LIN {X 0.123,Y -389.631,Z 435.593,A 0.000,B 0.000,C 90.000,E1 286.732} C_DIS
LIN {X -0.073,Y -402.281,Z 435.585,A 0.000,B 0.000,C 90.000,E1 285.371} C_DIS
LIN {X 0.165,Y -425.861,Z 435.572,A 0.000,B 0.000,C 90.000,E1 283.008} C_DIS
LIN {X -0.160,Y -433.525,Z 435.568,A 0.000,B 0.000,C 90.000,E1 282.299} C_DIS
LIN {X -0.184,Y -440.934,Z 435.564,A 0.000,B 0.000,C 90.000,E1 281.535} C_DIS
LIN {X 0.085,Y -448.117,Z 435.560,A 0.000,B 0.000,C 90.000,E1 280.715} C_DIS
LIN {X -0.168,Y -454.839,Z 435.555,A 0.000,B 0.000,C 90.000,E1 279.962} C_DIS
LIN {X 0.100,Y -461.020,Z 435.551,A 0.000,B 0.000,C 90.000,E1 279.151} C_DIS
LIN {X -0.034,Y -466.745,Z 435.547,A 0.000,B 0.000,C 90.000,E1 278.398} C_DIS
LIN {X 0.195,Y -473.496,Z 435.541,A 0.000,B 0.000,C 90.000,E1 277.352} C_DIS
LIN {X 0.113,Y -478.173,Z 435.537,A 0.000,B 0.000,C 90.000,E1 276.606} C_DIS
LIN {X 0.121,Y -482.372,Z 435.533,A 0.000,B 0.000,C 90.000,E1 275.853} C_DIS
LIN {X 0.118,Y -485.965,Z 435.528,A 0.000,B 0.000,C 90.000,E1 275.106} C_DIS
LIN {X 0.147,Y -488.810,Z 435.524,A 0.000,B 0.000,C 90.000,E1 274.359} C_DIS
LIN {X -0.139,Y -490.213,Z 435.522,A 0.000,B 0.000,C 90.000,E1 273.898} C_DIS
LIN {X 0.041,Y -491.202,Z 435.519,A 0.000,B 0.000,C 90.000,E1 273.383} C_DIS
LIN {X -0.232,Y -491.823,Z 435.516,A 0.000,B 0.000,C 90.000,E1 272.922} C_DIS
LIN {X -0.033,Y -492.111,Z 435.513,A 0.000,B 0.000,C 90.000,E1 272.407} C_DIS
LIN {X 0.172,Y -491.990,Z 435.511,A 0.000,B 0.000,C 90.000,E1 271.892} C_DIS
LIN {X -0.098,Y -491.492,Z 435.508,A 0.000,B 0.000,C 90.000,E1 271.432} C_DIS
LIN {X 0.107,Y -490.535,Z 435.505,A 0.000,B 0.000,C 90.000,E1 270.917} C_DIS
LIN {X -0.178,Y -489.067,Z 435.502,A 0.000,B 0.000,C 90.000,E1 270.458} C_DIS
LIN {X -0.128,Y -485.927,Z 435.498,A 0.000,B 0.000,C 90.000,E1 269.714} C_DIS
LIN {X 0.052,Y -483.029,Z 435.496,A 0.000,B 0.000,C 90.000,E1 269.198} C_DIS
LIN {X 0.210,Y -479.346,Z 435.493,A 0.000,B 0.000,C 90.000,E1 268.682} C_DIS
LIN {X -0.128,Y -474.646,Z 435.490,A 0.000,B 0.000,C 90.000,E1 268.224} C_DIS
LIN {X 0.188,Y -468.950,Z 435.487,A 0.000,B 0.000,C 90.000,E1 267.707} C_DIS
LIN {X -0.009,Y -462.615,Z 435.485,A 0.000,B 0.000,C 90.000,E1 267.306} C_DIS
LIN {X -0.137,Y -455.780,Z 435.483,A 0.000,B 0.000,C 90.000,E1 266.963} C_DIS
LIN {X -0.169,Y -448.676,Z 435.481,A 0.000,B 0.000,C 90.000,E1 266.674} C_DIS
LIN {X 0.179,Y -441.539,Z 435.480,A 0.000,B 0.000,C 90.000,E1 266.388} C_DIS
LIN {X -0.017,Y -433.742,Z 435.479,A 0.000,B 0.000,C 90.000,E1 266.216} C_DIS
LIN {X 0.183,Y -424.976,Z 435.478,A 0.000,B 0.000,C 90.000,E1 266.045} C_DIS
LIN {X -0.118,Y -414.468,Z 435.478,A 0.000,B 0.000,C 90.000,E1 265.988} C_DIS
LIN {X 0.107,Y -404.800,Z 435.477,A 0.000,B 0.000,C 90.000,E1 265.927} C_DIS
LIN {X 0.016,Y -180.918,Z 435.477,A 0.000,B 0.000,C 90.000,E1 265.927} C_DIS
LIN {X 0.049,Y -180.839,Z 435.472,A 0.000,B 0.000,C 90.000,E1 264.894} C_DIS
LIN {X -0.054,Y -178.880,Z 435.443,A 0.000,B 0.000,C 90.000,E1 259.690} C_DIS
LIN {X 0.022,Y -175.922,Z 435.414,A 0.000,B 0.000,C 90.000,E1 254.574} C_DIS
LIN {X -0.089,Y -174.621,Z 435.405,A 0.000,B 0.000,C 90.000,E1 252.906} C_DIS
LIN {X 0.004,Y -171.601,Z 435.381,A 0.000,B 0.000,C 90.000,E1 248.592} C_DIS
LIN {X -0.008,Y -167.824,Z 435.357,A 0.000,B 0.000,C 90.000,E1 244.280} C_DIS
LIN {X 0.010,Y -166.548,Z 435.347,A 0.000,B 0.000,C 90.000,E1 242.538} C_DIS
LIN {X -0.080,Y -162.545,Z 435.323,A 0.000,B 0.000,C 90.000,E1 238.201} C_DIS
LIN {X -0.019,Y -161.221,Z 435.313,A 0.000,B 0.000,C 90.000,E1 236.421} C_DIS
LIN {X 0.016,Y -157.229,Z 435.289,A 0.000,B 0.000,C 90.000,E1 231.984} C_DIS
LIN {X 0.039,Y -155.953,Z 435.279,A 0.000,B 0.000,C 90.000,E1 230.194} C_DIS
LIN {X -0.002,Y -152.206,Z 435.254,A 0.000,B 0.000,C 90.000,E1 225.729} C_DIS
LIN {X 0.018,Y -150.452,Z 435.239,A 0.000,B 0.000,C 90.000,E1 223.014} C_DIS
LIN {X 0.045,Y -147.177,Z 435.214,A 0.000,B 0.000,C 90.000,E1 218.463} C_DIS
LIN {X 0.012,Y -145.194,Z 435.193,A 0.000,B 0.000,C 90.000,E1 214.818} C_DIS
LIN {X 0.046,Y -142.335,Z 435.163,A 0.000,B 0.000,C 90.000,E1 209.283} C_DIS
LIN {X -0.025,Y -141.724,Z 435.153,A 0.000,B 0.000,C 90.000,E1 207.462} C_DIS
LIN {X -0.042,Y -139.478,Z 435.116,A 0.000,B 0.000,C 90.000,E1 200.972} C_DIS
LIN {X -0.054,Y -138.976,Z 435.101,A 0.000,B 0.000,C 90.000,E1 198.181} C_DIS
LIN {X 0.068,Y -138.332,Z 435.054,A 0.000,B 0.000,C 90.000,E1 189.726} C_DIS
LIN {X -0.068,Y -139.431,Z 435.007,A 0.000,B 0.000,C 90.000,E1 181.375} C_DIS
LIN {X 0.012,Y -140.958,Z 434.976,A 0.000,B 0.000,C 90.000,E1 175.755} C_DIS
LIN {X -0.038,Y -142.714,Z 434.956,A 0.000,B 0.000,C 90.000,E1 172.064} C_DIS
LIN {X 0.062,Y -145.091,Z 434.930,A 0.000,B 0.000,C 90.000,E1 167.409} C_DIS
LIN {X 0.057,Y -147.716,Z 434.910,A 0.000,B 0.000,C 90.000,E1 163.740} C_DIS
LIN {X -0.002,Y -150.372,Z 434.890,A 0.000,B 0.000,C 90.000,E1 160.115} C_DIS
LIN {X 0.016,Y -153.801,Z 434.869,A 0.000,B 0.000,C 90.000,E1 156.485} C_DIS
LIN {X 0.076,Y -157.213,Z 434.849,A 0.000,B 0.000,C 90.000,E1 152.871} C_DIS
LIN {X 0.017,Y -161.377,Z 434.830,A 0.000,B 0.000,C 90.000,E1 149.331} C_DIS
LIN {X 0.028,Y -165.580,Z 434.810,A 0.000,B 0.000,C 90.000,E1 145.801} C_DIS
LIN {X 0.015,Y -170.500,Z 434.791,A 0.000,B 0.000,C 90.000,E1 142.316} C_DIS
LIN {X 0.059,Y -175.380,Z 434.772,A 0.000,B 0.000,C 90.000,E1 138.852} C_DIS
LIN {X -0.079,Y -181.005,Z 434.753,A 0.000,B 0.000,C 90.000,E1 135.486} C_DIS
LIN {X 0.046,Y -186.434,Z 434.734,A 0.000,B 0.000,C 90.000,E1 132.081} C_DIS
LIN {X 0.115,Y -191.060,Z 434.720,A 0.000,B 0.000,C 90.000,E1 129.564} C_DIS
LIN {X 0.004,Y -195.867,Z 434.705,A 0.000,B 0.000,C 90.000,E1 126.824} C_DIS
LIN {X 0.135,Y -294.379,Z 434.705,A 0.000,B 0.000,C 90.000,E1 126.790} C_DIS
LIN {X -0.008,Y -296.001,Z 434.704,A 0.000,B 0.000,C 90.000,E1 126.790} C_DIS
LIN {X 0.056,Y -300.860,Z 434.703,A 0.000,B 0.000,C 90.000,E1 126.537} C_DIS
LIN {X 0.058,Y -303.494,Z 434.702,A 0.000,B 0.000,C 90.000,E1 126.297} C_DIS
LIN {X -0.117,Y -307.272,Z 434.699,A 0.000,B 0.000,C 90.000,E1 125.804} C_DIS
LIN {X 0.085,Y -308.927,Z 434.697,A 0.000,B 0.000,C 90.000,E1 125.438} C_DIS
LIN {X 0.109,Y -310.232,Z 434.695,A 0.000,B 0.000,C 90.000,E1 125.105} C_DIS
LIN {X -0.103,Y -322.084,Z 434.675,A 0.000,B 0.000,C 90.000,E1 121.592} C_DIS
LIN {X -0.105,Y -333.198,Z 434.660,A 0.000,B 0.000,C 90.000,E1 118.743} C_DIS
LIN {X 0.047,Y -345.725,Z 434.644,A 0.000,B 0.000,C 90.000,E1 115.924} C_DIS
LIN {X -0.096,Y -358.139,Z 434.631,A 0.000,B 0.000,C 90.000,E1 113.515} C_DIS
LIN {X 0.113,Y -371.851,Z 434.617,A 0.000,B 0.000,C 90.000,E1 111.099} C_DIS
LIN {X 0.056,Y -386.960,Z 434.604,A 0.000,B 0.000,C 90.000,E1 108.779} C_DIS
LIN {X 0.125,Y -403.577,Z 434.592,A 0.000,B 0.000,C 90.000,E1 106.496} C_DIS
LIN {X -0.010,Y -421.825,Z 434.579,A 0.000,B 0.000,C 90.000,E1 104.300} C_DIS
LIN {X -0.034,Y -441.588,Z 434.568,A 0.000,B 0.000,C 90.000,E1 102.175} C_DIS
LIN {X 0.112,Y -462.024,Z 434.557,A 0.000,B 0.000,C 90.000,E1 100.197} C_DIS
LIN {X -0.173,Y -485.514,Z 434.546,A 0.000,B 0.000,C 90.000,E1 98.219} C_DIS
LIN {X 0.009,Y -489.050,Z 434.543,A 0.000,B 0.000,C 90.000,E1 97.757} C_DIS
LIN {X -0.167,Y -490.369,Z 434.542,A 0.000,B 0.000,C 90.000,E1 97.530} C_DIS
LIN {X 0.207,Y -491.341,Z 434.540,A 0.000,B 0.000,C 90.000,E1 97.239} C_DIS
LIN {X -0.056,Y -492.420,Z 434.538,A 0.000,B 0.000,C 90.000,E1 96.777} C_DIS
LIN {X 0.177,Y -492.489,Z 434.535,A 0.000,B 0.000,C 90.000,E1 96.258} C_DIS
LIN {X -0.075,Y -491.558,Z 434.532,A 0.000,B 0.000,C 90.000,E1 95.796} C_DIS
LIN {X 0.161,Y -489.465,Z 434.529,A 0.000,B 0.000,C 90.000,E1 95.277} C_DIS
LIN {X 0.011,Y -487.840,Z 434.528,A 0.000,B 0.000,C 90.000,E1 95.049} C_DIS
LIN {X -0.226,Y -478.097,Z 434.521,A 0.000,B 0.000,C 90.000,E1 93.841} C_DIS
LIN {X 0.010,Y -456.548,Z 434.506,A 0.000,B 0.000,C 90.000,E1 91.031} C_DIS
LIN {X 0.172,Y -444.184,Z 434.496,A 0.000,B 0.000,C 90.000,E1 89.198} C_DIS
LIN {X -0.022,Y -429.185,Z 434.482,A 0.000,B 0.000,C 90.000,E1 86.846} C_DIS
LIN {X -0.046,Y -413.302,Z 434.467,A 0.000,B 0.000,C 90.000,E1 84.147} C_DIS
LIN {X -0.128,Y -400.978,Z 434.455,A 0.000,B 0.000,C 90.000,E1 81.951} C_DIS
LIN {X -0.101,Y -390.349,Z 434.444,A 0.000,B 0.000,C 90.000,E1 79.982} C_DIS
LIN {X 0.180,Y -381.300,Z 434.435,A 0.000,B 0.000,C 90.000,E1 78.229} C_DIS
LIN {X 0.081,Y -366.697,Z 434.419,A 0.000,B 0.000,C 90.000,E1 75.338} C_DIS
LIN {X 0.065,Y -350.448,Z 434.399,A 0.000,B 0.000,C 90.000,E1 71.764} C_DIS
LIN {X 0.015,Y -339.131,Z 434.384,A 0.000,B 0.000,C 90.000,E1 69.028} C_DIS
LIN {X 0.059,Y -329.454,Z 434.370,A 0.000,B 0.000,C 90.000,E1 66.538} C_DIS
LIN {X -0.056,Y -318.843,Z 434.354,A 0.000,B 0.000,C 90.000,E1 63.717} C_DIS
LIN {X 0.040,Y -309.658,Z 434.340,A 0.000,B 0.000,C 90.000,E1 61.129} C_DIS
LIN {X -0.012,Y -298.573,Z 434.321,A 0.000,B 0.000,C 90.000,E1 57.867} C_DIS
LIN {X 0.030,Y -288.435,Z 434.303,A 0.000,B 0.000,C 90.000,E1 54.529} C_DIS
LIN {X 0.017,Y -280.852,Z 434.288,A 0.000,B 0.000,C 90.000,E1 51.823} C_DIS
LIN {X 0.115,Y -275.170,Z 434.276,A 0.000,B 0.000,C 90.000,E1 49.747} C_DIS
LIN {X -0.105,Y -269.235,Z 434.265,A 0.000,B 0.000,C 90.000,E1 47.715} C_DIS
LIN {X 0.105,Y -263.070,Z 434.253,A 0.000,B 0.000,C 90.000,E1 45.567} C_DIS
LIN {X 0.012,Y -256.793,Z 434.241,A 0.000,B 0.000,C 90.000,E1 43.461} C_DIS
LIN {X 0.001,Y -250.333,Z 434.229,A 0.000,B 0.000,C 90.000,E1 41.310} C_DIS
LIN {X 0.045,Y -239.769,Z 434.209,A 0.000,B 0.000,C 90.000,E1 37.649} C_DIS
LIN {X -0.031,Y -231.877,Z 434.193,A 0.000,B 0.000,C 90.000,E1 34.692} C_DIS
LIN {X -0.045,Y -224.697,Z 434.176,A 0.000,B 0.000,C 90.000,E1 31.671} C_DIS
LIN {X -0.090,Y -218.311,Z 434.159,A 0.000,B 0.000,C 90.000,E1 28.615} C_DIS
LIN {X 0.069,Y -212.674,Z 434.142,A 0.000,B 0.000,C 90.000,E1 25.463} C_DIS
LIN {X 0.029,Y -206.563,Z 434.120,A 0.000,B 0.000,C 90.000,E1 21.535} C_DIS
LIN {X -0.102,Y -201.340,Z 434.098,A 0.000,B 0.000,C 90.000,E1 17.583} C_DIS
LIN {X -0.052,Y -197.150,Z 434.075,A 0.000,B 0.000,C 90.000,E1 13.536} C_DIS
LIN {X 0.032,Y -193.335,Z 434.048,A 0.000,B 0.000,C 90.000,E1 8.624} C_DIS
LIN {X -0.006,Y -190.457,Z 434.011,A 0.000,B 0.000,C 90.000,E1 2.064} C_DIS
LIN {X -0.008,Y -191.173,Z 433.961,A 0.000,B 0.000,C 90.000,E1 352.932} C_DIS
LIN {X 0.006,Y -194.242,Z 433.929,A 0.000,B 0.000,C 90.000,E1 347.173} C_DIS
LIN {X -0.103,Y -198.351,Z 433.902,A 0.000,B 0.000,C 90.000,E1 342.308} C_DIS
LIN {X 0.010,Y -202.852,Z 433.879,A 0.000,B 0.000,C 90.000,E1 338.230} C_DIS
LIN {X 0.006,Y -208.404,Z 433.857,A 0.000,B 0.000,C 90.000,E1 334.229} C_DIS
LIN {X 0.083,Y -214.790,Z 433.835,A 0.000,B 0.000,C 90.000,E1 330.255} C_DIS
LIN {X 0.018,Y -221.686,Z 433.813,A 0.000,B 0.000,C 90.000,E1 326.373} C_DIS
LIN {X -0.082,Y -229.246,Z 433.792,A 0.000,B 0.000,C 90.000,E1 322.557} C_DIS
LIN {X -0.060,Y -237.792,Z 433.771,A 0.000,B 0.000,C 90.000,E1 318.771} C_DIS
LIN {X 0.032,Y -246.477,Z 433.752,A 0.000,B 0.000,C 90.000,E1 315.405} C_DIS
LIN {X -0.148,Y -255.172,Z 433.736,A 0.000,B 0.000,C 90.000,E1 312.528} C_DIS
LIN {X -0.018,Y -266.116,Z 433.718,A 0.000,B 0.000,C 90.000,E1 309.277} C_DIS
LIN {X -0.072,Y -278.087,Z 433.701,A 0.000,B 0.000,C 90.000,E1 306.137} C_DIS
LIN {X 0.042,Y -289.473,Z 433.685,A 0.000,B 0.000,C 90.000,E1 303.372} C_DIS
LIN {X -0.084,Y -304.390,Z 433.667,A 0.000,B 0.000,C 90.000,E1 300.050} C_DIS
LIN {X -0.090,Y -320.673,Z 433.649,A 0.000,B 0.000,C 90.000,E1 296.796} C_DIS
LIN {X -0.121,Y -336.820,Z 433.633,A 0.000,B 0.000,C 90.000,E1 293.951} C_DIS
LIN {X 0.023,Y -353.039,Z 433.619,A 0.000,B 0.000,C 90.000,E1 291.461} C_DIS
LIN {X -0.137,Y -370.722,Z 433.606,A 0.000,B 0.000,C 90.000,E1 289.087} C_DIS
LIN {X 0.026,Y -389.759,Z 433.593,A 0.000,B 0.000,C 90.000,E1 286.732} C_DIS
LIN {X 0.144,Y -404.944,Z 433.584,A 0.000,B 0.000,C 90.000,E1 285.064} C_DIS
LIN {X 0.164,Y -425.900,Z 433.572,A 0.000,B 0.000,C 90.000,E1 283.008} C_DIS
LIN {X -0.156,Y -433.580,Z 433.568,A 0.000,B 0.000,C 90.000,E1 282.299} C_DIS
LIN {X 0.043,Y -443.390,Z 433.563,A 0.000,B 0.000,C 90.000,E1 281.243} C_DIS
LIN {X -0.227,Y -450.440,Z 433.558,A 0.000,B 0.000,C 90.000,E1 280.489} C_DIS
LIN {X 0.076,Y -456.998,Z 433.554,A 0.000,B 0.000,C 90.000,E1 279.670} C_DIS
LIN {X -0.096,Y -463.001,Z 433.549,A 0.000,B 0.000,C 90.000,E1 278.916} C_DIS
LIN {X -0.212,Y -468.492,Z 433.545,A 0.000,B 0.000,C 90.000,E1 278.163} C_DIS
LIN {X -0.028,Y -475.101,Z 433.540,A 0.000,B 0.000,C 90.000,E1 277.125} C_DIS
LIN {X -0.047,Y -479.630,Z 433.535,A 0.000,B 0.000,C 90.000,E1 276.372} C_DIS
LIN {X -0.075,Y -483.657,Z 433.531,A 0.000,B 0.000,C 90.000,E1 275.625} C_DIS
LIN {X -0.068,Y -487.018,Z 433.527,A 0.000,B 0.000,C 90.000,E1 274.878} C_DIS
LIN {X 0.131,Y -488.800,Z 433.524,A 0.000,B 0.000,C 90.000,E1 274.359} C_DIS
LIN {X -0.155,Y -490.188,Z 433.522,A 0.000,B 0.000,C 90.000,E1 273.898} C_DIS
LIN {X 0.026,Y -491.171,Z 433.519,A 0.000,B 0.000,C 90.000,E1 273.383} C_DIS
LIN {X 0.244,Y -491.813,Z 433.516,A 0.000,B 0.000,C 90.000,E1 272.865} C_DIS
LIN {X -0.049,Y -492.116,Z 433.513,A 0.000,B 0.000,C 90.000,E1 272.407} C_DIS
LIN {X 0.156,Y -492.028,Z 433.511,A 0.000,B 0.000,C 90.000,E1 271.892} C_DIS
LIN {X -0.114,Y -491.524,Z 433.508,A 0.000,B 0.000,C 90.000,E1 271.432} C_DIS
LIN {X 0.092,Y -490.557,Z 433.505,A 0.000,B 0.000,C 90.000,E1 270.917} C_DIS
LIN {X -0.194,Y -489.104,Z 433.502,A 0.000,B 0.000,C 90.000,E1 270.458} C_DIS
LIN {X 0.005,Y -487.130,Z 433.500,A 0.000,B 0.000,C 90.000,E1 269.943} C_DIS
LIN {X 0.194,Y -484.575,Z 433.497,A 0.000,B 0.000,C 90.000,E1 269.427} C_DIS
LIN {X -0.120,Y -481.344,Z 433.494,A 0.000,B 0.000,C 90.000,E1 268.969} C_DIS
LIN {X 0.031,Y -477.139,Z 433.491,A 0.000,B 0.000,C 90.000,E1 268.453} C_DIS
LIN {X -0.143,Y -474.692,Z 433.490,A 0.000,B 0.000,C 90.000,E1 268.224} C_DIS
LIN {X 0.172,Y -469.070,Z 433.487,A 0.000,B 0.000,C 90.000,E1 267.707} C_DIS
LIN {X 0.169,Y -465.857,Z 433.486,A 0.000,B 0.000,C 90.000,E1 267.478} C_DIS
LIN {X 0.214,Y -459.156,Z 433.484,A 0.000,B 0.000,C 90.000,E1 267.078} C_DIS
LIN {X -0.067,Y -452.119,Z 433.482,A 0.000,B 0.000,C 90.000,E1 266.788} C_DIS
LIN {X 0.105,Y -445.016,Z 433.481,A 0.000,B 0.000,C 90.000,E1 266.502} C_DIS
LIN {X 0.191,Y -437.456,Z 433.479,A 0.000,B 0.000,C 90.000,E1 266.274} C_DIS
LIN {X 0.206,Y -429.445,Z 433.478,A 0.000,B 0.000,C 90.000,E1 266.102} C_DIS
LIN {X 0.123,Y -418.947,Z 433.478,A 0.000,B 0.000,C 90.000,E1 265.988} C_DIS
LIN {X 0.134,Y -408.679,Z 433.477,A 0.000,B 0.000,C 90.000,E1 265.927} C_DIS
LIN {X 0.028,Y -180.917,Z 433.477,A 0.000,B 0.000,C 90.000,E1 265.927} C_DIS
LIN {X 0.059,Y -180.839,Z 433.472,A 0.000,B 0.000,C 90.000,E1 264.894} C_DIS
LIN {X -0.044,Y -178.881,Z 433.443,A 0.000,B 0.000,C 90.000,E1 259.690} C_DIS
LIN {X 0.033,Y -175.924,Z 433.414,A 0.000,B 0.000,C 90.000,E1 254.574} C_DIS
LIN {X -0.022,Y -175.361,Z 433.410,A 0.000,B 0.000,C 90.000,E1 253.740} C_DIS
LIN {X 0.037,Y -172.140,Z 433.386,A 0.000,B 0.000,C 90.000,E1 249.444} C_DIS
LIN {X 0.014,Y -171.604,Z 433.381,A 0.000,B 0.000,C 90.000,E1 248.592} C_DIS
LIN {X 0.002,Y -167.827,Z 433.357,A 0.000,B 0.000,C 90.000,E1 244.280} C_DIS
LIN {X 0.020,Y -166.552,Z 433.347,A 0.000,B 0.000,C 90.000,E1 242.538} C_DIS
LIN {X -0.070,Y -162.547,Z 433.323,A 0.000,B 0.000,C 90.000,E1 238.201} C_DIS
LIN {X -0.010,Y -161.225,Z 433.313,A 0.000,B 0.000,C 90.000,E1 236.421} C_DIS
LIN {X 0.025,Y -157.231,Z 433.289,A 0.000,B 0.000,C 90.000,E1 231.984} C_DIS
LIN {X 0.048,Y -155.955,Z 433.279,A 0.000,B 0.000,C 90.000,E1 230.194} C_DIS
LIN {X 0.007,Y -152.209,Z 433.254,A 0.000,B 0.000,C 90.000,E1 225.729} C_DIS
LIN {X 0.028,Y -150.454,Z 433.239,A 0.000,B 0.000,C 90.000,E1 223.014} C_DIS
LIN {X 0.054,Y -147.179,Z 433.214,A 0.000,B 0.000,C 90.000,E1 218.463} C_DIS
LIN {X 0.021,Y -145.197,Z 433.193,A 0.000,B 0.000,C 90.000,E1 214.818} C_DIS
LIN {X 0.056,Y -142.336,Z 433.163,A 0.000,B 0.000,C 90.000,E1 209.283} C_DIS
LIN {X -0.015,Y -141.724,Z 433.153,A 0.000,B 0.000,C 90.000,E1 207.462} C_DIS
LIN {X -0.033,Y -139.479,Z 433.116,A 0.000,B 0.000,C 90.000,E1 200.972} C_DIS
LIN {X -0.044,Y -138.977,Z 433.101,A 0.000,B 0.000,C 90.000,E1 198.181} C_DIS
LIN {X 0.077,Y -138.331,Z 433.054,A 0.000,B 0.000,C 90.000,E1 189.726} C_DIS
LIN {X -0.059,Y -139.431,Z 433.008,A 0.000,B 0.000,C 90.000,E1 181.375} C_DIS
LIN {X 0.020,Y -140.956,Z 432.976,A 0.000,B 0.000,C 90.000,E1 175.755} C_DIS
LIN {X -0.029,Y -142.713,Z 432.956,A 0.000,B 0.000,C 90.000,E1 172.064} C_DIS
LIN {X 0.070,Y -145.089,Z 432.930,A 0.000,B 0.000,C 90.000,E1 167.409} C_DIS
LIN {X 0.066,Y -147.713,Z 432.910,A 0.000,B 0.000,C 90.000,E1 163.740} C_DIS
LIN {X 0.008,Y -150.370,Z 432.890,A 0.000,B 0.000,C 90.000,E1 160.115} C_DIS
LIN {X 0.025,Y -153.797,Z 432.869,A 0.000,B 0.000,C 90.000,E1 156.485} C_DIS
LIN {X 0.086,Y -157.210,Z 432.849,A 0.000,B 0.000,C 90.000,E1 152.871} C_DIS
LIN {X 0.028,Y -161.373,Z 432.830,A 0.000,B 0.000,C 90.000,E1 149.331} C_DIS
LIN {X 0.039,Y -165.575,Z 432.810,A 0.000,B 0.000,C 90.000,E1 145.801} C_DIS
LIN {X 0.025,Y -170.495,Z 432.791,A 0.000,B 0.000,C 90.000,E1 142.316} C_DIS
LIN {X 0.070,Y -175.375,Z 432.772,A 0.000,B 0.000,C 90.000,E1 138.852} C_DIS
LIN {X -0.067,Y -180.999,Z 432.753,A 0.000,B 0.000,C 90.000,E1 135.486} C_DIS
LIN {X 0.057,Y -186.427,Z 432.734,A 0.000,B 0.000,C 90.000,E1 132.081} C_DIS
LIN {X 0.004,Y -191.054,Z 432.720,A 0.000,B 0.000,C 90.000,E1 129.600} C_DIS
LIN {X -0.067,Y -195.970,Z 432.704,A 0.000,B 0.000,C 90.000,E1 126.790} C_DIS
LIN {X -0.136,Y -294.358,Z 432.704,A 0.000,B 0.000,C 90.000,E1 126.790} C_DIS
LIN {X -0.078,Y -296.347,Z 432.704,A 0.000,B 0.000,C 90.000,E1 126.744} C_DIS
LIN {X 0.087,Y -300.646,Z 432.703,A 0.000,B 0.000,C 90.000,E1 126.503} C_DIS
LIN {X 0.076,Y -303.088,Z 432.702,A 0.000,B 0.000,C 90.000,E1 126.297} C_DIS
LIN {X 0.046,Y -306.923,Z 432.699,A 0.000,B 0.000,C 90.000,E1 125.804} C_DIS
LIN {X 0.067,Y -308.689,Z 432.697,A 0.000,B 0.000,C 90.000,E1 125.471} C_DIS
LIN {X 0.016,Y -310.075,Z 432.695,A 0.000,B 0.000,C 90.000,E1 125.152} C_DIS
LIN {X 0.059,Y -321.958,Z 432.676,A 0.000,B 0.000,C 90.000,E1 121.592} C_DIS
LIN {X 0.060,Y -333.058,Z 432.660,A 0.000,B 0.000,C 90.000,E1 118.743} C_DIS
LIN {X -0.098,Y -345.570,Z 432.644,A 0.000,B 0.000,C 90.000,E1 115.976} C_DIS
LIN {X 0.072,Y -357.970,Z 432.631,A 0.000,B 0.000,C 90.000,E1 113.515} C_DIS
LIN {X -0.062,Y -371.666,Z 432.617,A 0.000,B 0.000,C 90.000,E1 111.153} C_DIS
LIN {X 0.228,Y -386.759,Z 432.605,A 0.000,B 0.000,C 90.000,E1 108.779} C_DIS
LIN {X -0.088,Y -403.359,Z 432.592,A 0.000,B 0.000,C 90.000,E1 106.551} C_DIS
LIN {X 0.167,Y -421.587,Z 432.580,A 0.000,B 0.000,C 90.000,E1 104.300} C_DIS
LIN {X 0.045,Y -441.338,Z 432.568,A 0.000,B 0.000,C 90.000,E1 102.187} C_DIS
LIN {X -0.178,Y -461.768,Z 432.557,A 0.000,B 0.000,C 90.000,E1 100.254} C_DIS
LIN {X -0.017,Y -485.314,Z 432.546,A 0.000,B 0.000,C 90.000,E1 98.219} C_DIS
LIN {X 0.221,Y -488.968,Z 432.543,A 0.000,B 0.000,C 90.000,E1 97.757} C_DIS
LIN {X 0.045,Y -490.355,Z 432.542,A 0.000,B 0.000,C 90.000,E1 97.530} C_DIS
LIN {X -0.069,Y -491.381,Z 432.540,A 0.000,B 0.000,C 90.000,E1 97.296} C_DIS
LIN {X 0.156,Y -492.551,Z 432.538,A 0.000,B 0.000,C 90.000,E1 96.777} C_DIS
LIN {X -0.101,Y -492.701,Z 432.535,A 0.000,B 0.000,C 90.000,E1 96.315} C_DIS
LIN {X 0.138,Y -491.856,Z 432.532,A 0.000,B 0.000,C 90.000,E1 95.796} C_DIS
LIN {X -0.113,Y -489.871,Z 432.530,A 0.000,B 0.000,C 90.000,E1 95.334} C_DIS
LIN {X 0.223,Y -488.323,Z 432.528,A 0.000,B 0.000,C 90.000,E1 95.049} C_DIS
LIN {X -0.011,Y -478.613,Z 432.521,A 0.000,B 0.000,C 90.000,E1 93.841} C_DIS
LIN {X -0.225,Y -457.032,Z 432.506,A 0.000,B 0.000,C 90.000,E1 91.088} C_DIS
LIN {X -0.048,Y -444.611,Z 432.496,A 0.000,B 0.000,C 90.000,E1 89.255} C_DIS
LIN {X 0.182,Y -429.586,Z 432.483,A 0.000,B 0.000,C 90.000,E1 86.849} C_DIS
LIN {X 0.184,Y -413.679,Z 432.468,A 0.000,B 0.000,C 90.000,E1 84.147} C_DIS
LIN {X 0.105,Y -401.363,Z 432.455,A 0.000,B 0.000,C 90.000,E1 81.951} C_DIS
LIN {X 0.133,Y -390.733,Z 432.444,A 0.000,B 0.000,C 90.000,E1 79.982} C_DIS
LIN {X 0.072,Y -380.174,Z 432.433,A 0.000,B 0.000,C 90.000,E1 77.993} C_DIS
LIN {X -0.053,Y -365.677,Z 432.417,A 0.000,B 0.000,C 90.000,E1 75.102} C_DIS
LIN {X 0.008,Y -349.513,Z 432.397,A 0.000,B 0.000,C 90.000,E1 71.511} C_DIS
LIN {X -0.053,Y -338.211,Z 432.382,A 0.000,B 0.000,C 90.000,E1 68.773} C_DIS
LIN {X -0.155,Y -328.526,Z 432.368,A 0.000,B 0.000,C 90.000,E1 66.305} C_DIS
LIN {X -0.098,Y -319.068,Z 432.354,A 0.000,B 0.000,C 90.000,E1 63.768} C_DIS
LIN {X 0.010,Y -309.854,Z 432.340,A 0.000,B 0.000,C 90.000,E1 61.179} C_DIS
LIN {X -0.026,Y -298.738,Z 432.322,A 0.000,B 0.000,C 90.000,E1 57.916} C_DIS
LIN {X 0.099,Y -288.582,Z 432.303,A 0.000,B 0.000,C 90.000,E1 54.562} C_DIS
LIN {X -0.145,Y -280.976,Z 432.288,A 0.000,B 0.000,C 90.000,E1 51.904} C_DIS
LIN {X -0.043,Y -275.316,Z 432.277,A 0.000,B 0.000,C 90.000,E1 49.828} C_DIS
LIN {X -0.077,Y -269.405,Z 432.265,A 0.000,B 0.000,C 90.000,E1 47.757} C_DIS
LIN {X -0.041,Y -263.266,Z 432.254,A 0.000,B 0.000,C 90.000,E1 45.648} C_DIS
LIN {X -0.127,Y -257.002,Z 432.242,A 0.000,B 0.000,C 90.000,E1 43.542} C_DIS
LIN {X 0.035,Y -250.558,Z 432.230,A 0.000,B 0.000,C 90.000,E1 41.353} C_DIS
LIN {X -0.071,Y -239.971,Z 432.210,A 0.000,B 0.000,C 90.000,E1 37.729} C_DIS
LIN {X -0.005,Y -232.074,Z 432.193,A 0.000,B 0.000,C 90.000,E1 34.739} C_DIS
LIN {X -0.020,Y -224.884,Z 432.176,A 0.000,B 0.000,C 90.000,E1 31.720} C_DIS
LIN {X 0.124,Y -218.481,Z 432.159,A 0.000,B 0.000,C 90.000,E1 28.615} C_DIS
LIN {X -0.003,Y -212.810,Z 432.142,A 0.000,B 0.000,C 90.000,E1 25.540} C_DIS
LIN {X 0.048,Y -206.652,Z 432.120,A 0.000,B 0.000,C 90.000,E1 21.589} C_DIS
LIN {X -0.087,Y -201.397,Z 432.098,A 0.000,B 0.000,C 90.000,E1 17.638} C_DIS
LIN {X -0.039,Y -197.171,Z 432.075,A 0.000,B 0.000,C 90.000,E1 13.592} C_DIS
LIN {X 0.042,Y -193.299,Z 432.048,A 0.000,B 0.000,C 90.000,E1 8.681} C_DIS
LIN {X 0.000,Y -190.373,Z 432.012,A 0.000,B 0.000,C 90.000,E1 2.121} C_DIS
LIN {X -0.014,Y -191.050,Z 431.961,A 0.000,B 0.000,C 90.000,E1 352.932} C_DIS
LIN {X -0.005,Y -194.109,Z 431.929,A 0.000,B 0.000,C 90.000,E1 347.173} C_DIS
LIN {X -0.119,Y -198.201,Z 431.902,A 0.000,B 0.000,C 90.000,E1 342.308} C_DIS
LIN {X -0.011,Y -202.692,Z 431.879,A 0.000,B 0.000,C 90.000,E1 338.230} C_DIS
LIN {X 0.070,Y -208.248,Z 431.857,A 0.000,B 0.000,C 90.000,E1 334.204} C_DIS
LIN {X 0.049,Y -214.655,Z 431.835,A 0.000,B 0.000,C 90.000,E1 330.255} C_DIS
LIN {X -0.020,Y -221.535,Z 431.813,A 0.000,B 0.000,C 90.000,E1 326.373} C_DIS
LIN {X -0.126,Y -229.093,Z 431.792,A 0.000,B 0.000,C 90.000,E1 322.557} C_DIS
LIN {X -0.111,Y -237.665,Z 431.771,A 0.000,B 0.000,C 90.000,E1 318.771} C_DIS
LIN {X -0.024,Y -246.355,Z 431.752,A 0.000,B 0.000,C 90.000,E1 315.405} C_DIS
LIN {X -0.021,Y -255.067,Z 431.736,A 0.000,B 0.000,C 90.000,E1 312.486} C_DIS
LIN {X -0.085,Y -266.038,Z 431.718,A 0.000,B 0.000,C 90.000,E1 309.277} C_DIS
LIN {X -0.018,Y -276.665,Z 431.703,A 0.000,B 0.000,C 90.000,E1 306.457} C_DIS
LIN {X -0.006,Y -287.995,Z 431.687,A 0.000,B 0.000,C 90.000,E1 303.706} C_DIS
LIN {X 0.077,Y -302.843,Z 431.669,A 0.000,B 0.000,C 90.000,E1 300.335} C_DIS
LIN {X 0.041,Y -318.949,Z 431.650,A 0.000,B 0.000,C 90.000,E1 297.078} C_DIS
LIN {X 0.125,Y -334.957,Z 431.635,A 0.000,B 0.000,C 90.000,E1 294.207} C_DIS
LIN {X -0.110,Y -348.920,Z 431.623,A 0.000,B 0.000,C 90.000,E1 292.078} C_DIS
LIN {X 0.164,Y -368.504,Z 431.607,A 0.000,B 0.000,C 90.000,E1 289.322} C_DIS
LIN {X -0.070,Y -389.876,Z 431.593,A 0.000,B 0.000,C 90.000,E1 286.732} C_DIS
LIN {X -0.036,Y -405.222,Z 431.584,A 0.000,B 0.000,C 90.000,E1 285.064} C_DIS
LIN {X 0.055,Y -423.624,Z 431.574,A 0.000,B 0.000,C 90.000,E1 283.244} C_DIS
LIN {X 0.151,Y -431.418,Z 431.569,A 0.000,B 0.000,C 90.000,E1 282.479} C_DIS
LIN {X 0.144,Y -438.892,Z 431.565,A 0.000,B 0.000,C 90.000,E1 281.715} C_DIS
LIN {X -0.012,Y -446.170,Z 431.561,A 0.000,B 0.000,C 90.000,E1 280.950} C_DIS
LIN {X 0.082,Y -455.135,Z 431.555,A 0.000,B 0.000,C 90.000,E1 279.905} C_DIS
LIN {X -0.098,Y -461.267,Z 431.551,A 0.000,B 0.000,C 90.000,E1 279.151} C_DIS
LIN {X 0.068,Y -468.634,Z 431.545,A 0.000,B 0.000,C 90.000,E1 278.106} C_DIS
LIN {X -0.213,Y -475.234,Z 431.539,A 0.000,B 0.000,C 90.000,E1 277.125} C_DIS
LIN {X -0.232,Y -479.753,Z 431.535,A 0.000,B 0.000,C 90.000,E1 276.372} C_DIS
LIN {X 0.222,Y -483.765,Z 431.531,A 0.000,B 0.000,C 90.000,E1 275.568} C_DIS
LIN {X -0.083,Y -486.062,Z 431.528,A 0.000,B 0.000,C 90.000,E1 275.106} C_DIS
LIN {X -0.254,Y -487.090,Z 431.527,A 0.000,B 0.000,C 90.000,E1 274.878} C_DIS
LIN {X -0.056,Y -488.822,Z 431.524,A 0.000,B 0.000,C 90.000,E1 274.359} C_DIS
LIN {X 0.147,Y -490.203,Z 431.521,A 0.000,B 0.000,C 90.000,E1 273.841} C_DIS
LIN {X -0.162,Y -491.184,Z 431.519,A 0.000,B 0.000,C 90.000,E1 273.383} C_DIS
LIN {X 0.056,Y -491.840,Z 431.516,A 0.000,B 0.000,C 90.000,E1 272.865} C_DIS
LIN {X -0.236,Y -492.126,Z 431.513,A 0.000,B 0.000,C 90.000,E1 272.407} C_DIS
LIN {X -0.031,Y -492.005,Z 431.510,A 0.000,B 0.000,C 90.000,E1 271.892} C_DIS
LIN {X 0.190,Y -491.517,Z 431.508,A 0.000,B 0.000,C 90.000,E1 271.375} C_DIS
LIN {X -0.095,Y -490.546,Z 431.505,A 0.000,B 0.000,C 90.000,E1 270.917} C_DIS
LIN {X 0.110,Y -489.059,Z 431.502,A 0.000,B 0.000,C 90.000,E1 270.401} C_DIS
LIN {X -0.180,Y -487.079,Z 431.500,A 0.000,B 0.000,C 90.000,E1 269.943} C_DIS
LIN {X 0.010,Y -484.491,Z 431.497,A 0.000,B 0.000,C 90.000,E1 269.427} C_DIS
LIN {X 0.177,Y -481.206,Z 431.494,A 0.000,B 0.000,C 90.000,E1 268.912} C_DIS
LIN {X -0.151,Y -477.016,Z 431.491,A 0.000,B 0.000,C 90.000,E1 268.453} C_DIS
LIN {X 0.165,Y -474.539,Z 431.490,A 0.000,B 0.000,C 90.000,E1 268.165} C_DIS
LIN {X -0.001,Y -468.873,Z 431.487,A 0.000,B 0.000,C 90.000,E1 267.707} C_DIS
LIN {X 0.005,Y -465.673,Z 431.486,A 0.000,B 0.000,C 90.000,E1 267.478} C_DIS
LIN {X 0.054,Y -458.961,Z 431.484,A 0.000,B 0.000,C 90.000,E1 267.078} C_DIS
LIN {X 0.225,Y -451.780,Z 431.482,A 0.000,B 0.000,C 90.000,E1 266.731} C_DIS
LIN {X -0.018,Y -444.635,Z 431.481,A 0.000,B 0.000,C 90.000,E1 266.502} C_DIS
LIN {X 0.118,Y -437.225,Z 431.479,A 0.000,B 0.000,C 90.000,E1 266.274} C_DIS
LIN {X 0.148,Y -429.031,Z 431.478,A 0.000,B 0.000,C 90.000,E1 266.102} C_DIS
LIN {X 0.084,Y -418.453,Z 431.478,A 0.000,B 0.000,C 90.000,E1 265.988} C_DIS
LIN {X 0.103,Y -406.272,Z 431.477,A 0.000,B 0.000,C 90.000,E1 265.927} C_DIS
LIN {X 0.015,Y -180.917,Z 431.477,A 0.000,B 0.000,C 90.000,E1 265.927} C_DIS
LIN {X 0.047,Y -180.838,Z 431.472,A 0.000,B 0.000,C 90.000,E1 264.894} C_DIS
LIN {X -0.055,Y -178.879,Z 431.443,A 0.000,B 0.000,C 90.000,E1 259.690} C_DIS
LIN {X 0.021,Y -175.922,Z 431.414,A 0.000,B 0.000,C 90.000,E1 254.574} C_DIS
LIN {X -0.090,Y -174.621,Z 431.405,A 0.000,B 0.000,C 90.000,E1 252.906} C_DIS
LIN {X 0.002,Y -171.601,Z 431.381,A 0.000,B 0.000,C 90.000,E1 248.592} C_DIS
LIN {X -0.009,Y -167.823,Z 431.357,A 0.000,B 0.000,C 90.000,E1 244.280} C_DIS
LIN {X 0.009,Y -166.547,Z 431.347,A 0.000,B 0.000,C 90.000,E1 242.538} C_DIS
LIN {X -0.081,Y -162.544,Z 431.323,A 0.000,B 0.000,C 90.000,E1 238.201} C_DIS
LIN {X -0.021,Y -161.221,Z 431.313,A 0.000,B 0.000,C 90.000,E1 236.421} C_DIS
LIN {X 0.015,Y -157.228,Z 431.289,A 0.000,B 0.000,C 90.000,E1 231.984} C_DIS
LIN {X 0.037,Y -155.953,Z 431.279,A 0.000,B 0.000,C 90.000,E1 230.194} C_DIS
LIN {X -0.003,Y -152.206,Z 431.254,A 0.000,B 0.000,C 90.000,E1 225.729} C_DIS
LIN {X 0.018,Y -150.451,Z 431.239,A 0.000,B 0.000,C 90.000,E1 223.014} C_DIS
LIN {X 0.044,Y -147.177,Z 431.214,A 0.000,B 0.000,C 90.000,E1 218.463} C_DIS
LIN {X 0.011,Y -145.194,Z 431.193,A 0.000,B 0.000,C 90.000,E1 214.818} C_DIS
LIN {X 0.045,Y -142.334,Z 431.163,A 0.000,B 0.000,C 90.000,E1 209.283} C_DIS
LIN {X -0.026,Y -141.723,Z 431.152,A 0.000,B 0.000,C 90.000,E1 207.462} C_DIS
LIN {X -0.043,Y -139.478,Z 431.116,A 0.000,B 0.000,C 90.000,E1 200.972} C_DIS
LIN {X -0.054,Y -138.975,Z 431.101,A 0.000,B 0.000,C 90.000,E1 198.181} C_DIS
LIN {X 0.067,Y -138.332,Z 431.054,A 0.000,B 0.000,C 90.000,E1 189.726} C_DIS
LIN {X 0.070,Y -139.431,Z 431.007,A 0.000,B 0.000,C 90.000,E1 181.318} C_DIS
LIN {X 0.011,Y -140.958,Z 430.976,A 0.000,B 0.000,C 90.000,E1 175.755} C_DIS
LIN {X -0.039,Y -142.714,Z 430.956,A 0.000,B 0.000,C 90.000,E1 172.064} C_DIS
LIN {X 0.060,Y -145.091,Z 430.930,A 0.000,B 0.000,C 90.000,E1 167.409} C_DIS
LIN {X 0.056,Y -147.716,Z 430.910,A 0.000,B 0.000,C 90.000,E1 163.740} C_DIS
LIN {X -0.003,Y -150.373,Z 430.890,A 0.000,B 0.000,C 90.000,E1 160.115} C_DIS
LIN {X 0.014,Y -153.802,Z 430.869,A 0.000,B 0.000,C 90.000,E1 156.485} C_DIS
LIN {X 0.075,Y -157.214,Z 430.849,A 0.000,B 0.000,C 90.000,E1 152.871} C_DIS
LIN {X 0.015,Y -161.378,Z 430.830,A 0.000,B 0.000,C 90.000,E1 149.331} C_DIS
LIN {X 0.027,Y -165.581,Z 430.810,A 0.000,B 0.000,C 90.000,E1 145.801} C_DIS
LIN {X 0.013,Y -170.501,Z 430.791,A 0.000,B 0.000,C 90.000,E1 142.316} C_DIS
LIN {X 0.058,Y -175.381,Z 430.772,A 0.000,B 0.000,C 90.000,E1 138.852} C_DIS
LIN {X -0.079,Y -181.005,Z 430.753,A 0.000,B 0.000,C 90.000,E1 135.486} C_DIS
LIN {X 0.045,Y -186.434,Z 430.734,A 0.000,B 0.000,C 90.000,E1 132.081} C_DIS
LIN {X 0.114,Y -191.060,Z 430.720,A 0.000,B 0.000,C 90.000,E1 129.564} C_DIS
LIN {X 0.026,Y -196.069,Z 430.704,A 0.000,B 0.000,C 90.000,E1 126.710} C_DIS
LIN {X 0.005,Y -294.502,Z 430.704,A 0.000,B 0.000,C 90.000,E1 126.710} C_DIS
LIN {X 0.032,Y -296.717,Z 430.704,A 0.000,B 0.000,C 90.000,E1 126.664} C_DIS
LIN {X -0.076,Y -300.492,Z 430.703,A 0.000,B 0.000,C 90.000,E1 126.503} C_DIS
LIN {X 0.056,Y -302.740,Z 430.702,A 0.000,B 0.000,C 90.000,E1 126.297} C_DIS
LIN {X 0.154,Y -306.618,Z 430.699,A 0.000,B 0.000,C 90.000,E1 125.804} C_DIS
LIN {X -0.071,Y -308.478,Z 430.697,A 0.000,B 0.000,C 90.000,E1 125.518} C_DIS
LIN {X -0.044,Y -309.932,Z 430.695,A 0.000,B 0.000,C 90.000,E1 125.185} C_DIS
LIN {X -0.144,Y -315.201,Z 430.686,A 0.000,B 0.000,C 90.000,E1 123.579} C_DIS
LIN {X -0.005,Y -325.406,Z 430.670,A 0.000,B 0.000,C 90.000,E1 120.669} C_DIS
LIN {X -0.060,Y -336.953,Z 430.655,A 0.000,B 0.000,C 90.000,E1 117.847} C_DIS
LIN {X -0.111,Y -349.952,Z 430.639,A 0.000,B 0.000,C 90.000,E1 115.079} C_DIS
LIN {X 0.023,Y -362.817,Z 430.626,A 0.000,B 0.000,C 90.000,E1 112.642} C_DIS
LIN {X -0.130,Y -377.013,Z 430.613,A 0.000,B 0.000,C 90.000,E1 110.301} C_DIS
LIN {X -0.196,Y -392.646,Z 430.600,A 0.000,B 0.000,C 90.000,E1 108.000} C_DIS
LIN {X 0.008,Y -409.828,Z 430.587,A 0.000,B 0.000,C 90.000,E1 105.717} C_DIS
LIN {X -0.085,Y -428.689,Z 430.575,A 0.000,B 0.000,C 90.000,E1 103.536} C_DIS
LIN {X -0.211,Y -448.758,Z 430.564,A 0.000,B 0.000,C 90.000,E1 101.478} C_DIS
LIN {X -0.038,Y -469.384,Z 430.553,A 0.000,B 0.000,C 90.000,E1 99.557} C_DIS
LIN {X 0.096,Y -485.152,Z 430.546,A 0.000,B 0.000,C 90.000,E1 98.219} C_DIS
LIN {X -0.117,Y -488.922,Z 430.543,A 0.000,B 0.000,C 90.000,E1 97.814} C_DIS
LIN {X 0.191,Y -490.363,Z 430.542,A 0.000,B 0.000,C 90.000,E1 97.530} C_DIS
LIN {X 0.077,Y -491.433,Z 430.541,A 0.000,B 0.000,C 90.000,E1 97.296} C_DIS
LIN {X -0.186,Y -492.670,Z 430.538,A 0.000,B 0.000,C 90.000,E1 96.834} C_DIS
LIN {X 0.046,Y -492.881,Z 430.535,A 0.000,B 0.000,C 90.000,E1 96.315} C_DIS
LIN {X -0.205,Y -492.101,Z 430.532,A 0.000,B 0.000,C 90.000,E1 95.853} C_DIS
LIN {X 0.034,Y -490.196,Z 430.530,A 0.000,B 0.000,C 90.000,E1 95.334} C_DIS
LIN {X -0.115,Y -488.703,Z 430.528,A 0.000,B 0.000,C 90.000,E1 95.106} C_DIS
LIN {X -0.211,Y -481.037,Z 430.523,A 0.000,B 0.000,C 90.000,E1 94.131} C_DIS
LIN {X -0.176,Y -465.122,Z 430.512,A 0.000,B 0.000,C 90.000,E1 92.121} C_DIS
LIN {X 0.173,Y -451.971,Z 430.502,A 0.000,B 0.000,C 90.000,E1 90.286} C_DIS
LIN {X 0.048,Y -433.226,Z 430.486,A 0.000,B 0.000,C 90.000,E1 87.421} C_DIS
LIN {X -0.146,Y -415.573,Z 430.469,A 0.000,B 0.000,C 90.000,E1 84.489} C_DIS
LIN {X 0.184,Y -403.231,Z 430.457,A 0.000,B 0.000,C 90.000,E1 82.243} C_DIS
LIN {X -0.145,Y -392.592,Z 430.446,A 0.000,B 0.000,C 90.000,E1 80.330} C_DIS
LIN {X -0.156,Y -382.036,Z 430.435,A 0.000,B 0.000,C 90.000,E1 78.342} C_DIS
LIN {X 0.050,Y -367.444,Z 430.419,A 0.000,B 0.000,C 90.000,E1 75.408} C_DIS
LIN {X 0.157,Y -351.137,Z 430.399,A 0.000,B 0.000,C 90.000,E1 71.819} C_DIS
LIN {X 0.127,Y -339.733,Z 430.384,A 0.000,B 0.000,C 90.000,E1 69.082} C_DIS
LIN {X 0.057,Y -329.967,Z 430.370,A 0.000,B 0.000,C 90.000,E1 66.613} C_DIS
LIN {X 0.005,Y -320.440,Z 430.356,A 0.000,B 0.000,C 90.000,E1 64.101} C_DIS
LIN {X 0.197,Y -310.014,Z 430.340,A 0.000,B 0.000,C 90.000,E1 61.179} C_DIS
LIN {X -0.001,Y -298.859,Z 430.322,A 0.000,B 0.000,C 90.000,E1 57.946} C_DIS
LIN {X 0.039,Y -288.691,Z 430.303,A 0.000,B 0.000,C 90.000,E1 54.609} C_DIS
LIN {X 0.028,Y -281.074,Z 430.288,A 0.000,B 0.000,C 90.000,E1 51.904} C_DIS
LIN {X 0.128,Y -275.420,Z 430.277,A 0.000,B 0.000,C 90.000,E1 49.828} C_DIS
LIN {X -0.089,Y -269.540,Z 430.265,A 0.000,B 0.000,C 90.000,E1 47.796} C_DIS
LIN {X 0.127,Y -263.423,Z 430.254,A 0.000,B 0.000,C 90.000,E1 45.648} C_DIS
LIN {X 0.039,Y -257.177,Z 430.242,A 0.000,B 0.000,C 90.000,E1 43.542} C_DIS
LIN {X 0.035,Y -250.748,Z 430.230,A 0.000,B 0.000,C 90.000,E1 41.391} C_DIS
LIN {X 0.094,Y -240.135,Z 430.210,A 0.000,B 0.000,C 90.000,E1 37.729} C_DIS
LIN {X 0.027,Y -232.237,Z 430.193,A 0.000,B 0.000,C 90.000,E1 34.771} C_DIS
LIN {X 0.024,Y -225.042,Z 430.176,A 0.000,B 0.000,C 90.000,E1 31.750} C_DIS
LIN {X -0.011,Y -218.629,Z 430.159,A 0.000,B 0.000,C 90.000,E1 28.693} C_DIS
LIN {X -0.033,Y -212.925,Z 430.142,A 0.000,B 0.000,C 90.000,E1 25.591} C_DIS
LIN {X -0.061,Y -206.733,Z 430.120,A 0.000,B 0.000,C 90.000,E1 21.663} C_DIS
LIN {X 0.071,Y -201.447,Z 430.098,A 0.000,B 0.000,C 90.000,E1 17.638} C_DIS
LIN {X -0.075,Y -197.187,Z 430.076,A 0.000,B 0.000,C 90.000,E1 13.647} C_DIS
LIN {X -0.025,Y -193.257,Z 430.049,A 0.000,B 0.000,C 90.000,E1 8.746} C_DIS
LIN {X -0.043,Y -190.295,Z 430.012,A 0.000,B 0.000,C 90.000,E1 2.178} C_DIS
LIN {X -0.091,Y -191.278,Z 429.956,A 0.000,B 0.000,C 90.000,E1 352.129} C_DIS
LIN {X -0.012,Y -194.572,Z 429.924,A 0.000,B 0.000,C 90.000,E1 346.353} C_DIS
LIN {X 0.114,Y -198.058,Z 429.901,A 0.000,B 0.000,C 90.000,E1 342.236} C_DIS
LIN {X -0.031,Y -202.538,Z 429.879,A 0.000,B 0.000,C 90.000,E1 338.230} C_DIS
LIN {X 0.044,Y -208.095,Z 429.857,A 0.000,B 0.000,C 90.000,E1 334.204} C_DIS
LIN {X 0.018,Y -214.508,Z 429.835,A 0.000,B 0.000,C 90.000,E1 330.255} C_DIS
LIN {X -0.057,Y -221.400,Z 429.813,A 0.000,B 0.000,C 90.000,E1 326.373} C_DIS
LIN {X 0.012,Y -228.941,Z 429.792,A 0.000,B 0.000,C 90.000,E1 322.512} C_DIS
LIN {X 0.019,Y -237.547,Z 429.771,A 0.000,B 0.000,C 90.000,E1 318.728} C_DIS
LIN {X -0.078,Y -246.250,Z 429.752,A 0.000,B 0.000,C 90.000,E1 315.405} C_DIS
LIN {X -0.099,Y -253.794,Z 429.738,A 0.000,B 0.000,C 90.000,E1 312.852} C_DIS
LIN {X 0.169,Y -264.666,Z 429.720,A 0.000,B 0.000,C 90.000,E1 309.564} C_DIS
LIN {X -0.011,Y -275.254,Z 429.704,A 0.000,B 0.000,C 90.000,E1 306.790} C_DIS
LIN {X -0.080,Y -287.962,Z 429.687,A 0.000,B 0.000,C 90.000,E1 303.706} C_DIS
LIN {X -0.012,Y -301.263,Z 429.670,A 0.000,B 0.000,C 90.000,E1 300.669} C_DIS
LIN {X 0.045,Y -317.243,Z 429.652,A 0.000,B 0.000,C 90.000,E1 297.385} C_DIS
LIN {X 0.037,Y -334.980,Z 429.635,A 0.000,B 0.000,C 90.000,E1 294.207} C_DIS
LIN {X 0.168,Y -353.197,Z 429.619,A 0.000,B 0.000,C 90.000,E1 291.408} C_DIS
LIN {X 0.071,Y -368.641,Z 429.607,A 0.000,B 0.000,C 90.000,E1 289.322} C_DIS
LIN {X -0.086,Y -389.913,Z 429.593,A 0.000,B 0.000,C 90.000,E1 286.732} C_DIS
LIN {X 0.122,Y -404.891,Z 429.584,A 0.000,B 0.000,C 90.000,E1 285.079} C_DIS
LIN {X -0.065,Y -423.283,Z 429.574,A 0.000,B 0.000,C 90.000,E1 283.300} C_DIS
LIN {X -0.117,Y -433.607,Z 429.568,A 0.000,B 0.000,C 90.000,E1 282.299} C_DIS
LIN {X 0.183,Y -443.310,Z 429.563,A 0.000,B 0.000,C 90.000,E1 281.243} C_DIS
LIN {X -0.179,Y -452.525,Z 429.557,A 0.000,B 0.000,C 90.000,E1 280.254} C_DIS
LIN {X 0.060,Y -458.856,Z 429.552,A 0.000,B 0.000,C 90.000,E1 279.443} C_DIS
LIN {X 0.202,Y -466.507,Z 429.547,A 0.000,B 0.000,C 90.000,E1 278.398} C_DIS
LIN {X -0.037,Y -473.294,Z 429.541,A 0.000,B 0.000,C 90.000,E1 277.409} C_DIS
LIN {X 0.207,Y -479.459,Z 429.536,A 0.000,B 0.000,C 90.000,E1 276.372} C_DIS
LIN {X 0.179,Y -483.489,Z 429.531,A 0.000,B 0.000,C 90.000,E1 275.625} C_DIS
LIN {X 0.186,Y -486.882,Z 429.527,A 0.000,B 0.000,C 90.000,E1 274.878} C_DIS
LIN {X -0.102,Y -488.659,Z 429.524,A 0.000,B 0.000,C 90.000,E1 274.416} C_DIS
LIN {X 0.099,Y -490.051,Z 429.522,A 0.000,B 0.000,C 90.000,E1 273.898} C_DIS
LIN {X -0.211,Y -491.070,Z 429.519,A 0.000,B 0.000,C 90.000,E1 273.440} C_DIS
LIN {X 0.006,Y -491.786,Z 429.516,A 0.000,B 0.000,C 90.000,E1 272.922} C_DIS
LIN {X 0.204,Y -492.113,Z 429.514,A 0.000,B 0.000,C 90.000,E1 272.407} C_DIS
LIN {X -0.083,Y -492.081,Z 429.511,A 0.000,B 0.000,C 90.000,E1 271.949} C_DIS
LIN {X 0.138,Y -491.617,Z 429.508,A 0.000,B 0.000,C 90.000,E1 271.432} C_DIS
LIN {X -0.147,Y -490.688,Z 429.505,A 0.000,B 0.000,C 90.000,E1 270.974} C_DIS
LIN {X 0.059,Y -489.271,Z 429.503,A 0.000,B 0.000,C 90.000,E1 270.458} C_DIS
LIN {X -0.230,Y -487.357,Z 429.500,A 0.000,B 0.000,C 90.000,E1 270.000} C_DIS
LIN {X -0.040,Y -484.843,Z 429.497,A 0.000,B 0.000,C 90.000,E1 269.484} C_DIS
LIN {X 0.131,Y -481.647,Z 429.494,A 0.000,B 0.000,C 90.000,E1 268.969} C_DIS
LIN {X -0.195,Y -477.565,Z 429.492,A 0.000,B 0.000,C 90.000,E1 268.511} C_DIS
LIN {X -0.048,Y -472.447,Z 429.489,A 0.000,B 0.000,C 90.000,E1 267.993} C_DIS
LIN {X -0.112,Y -469.571,Z 429.488,A 0.000,B 0.000,C 90.000,E1 267.764} C_DIS
LIN {X -0.175,Y -466.331,Z 429.486,A 0.000,B 0.000,C 90.000,E1 267.535} C_DIS
LIN {X -0.182,Y -459.590,Z 429.484,A 0.000,B 0.000,C 90.000,E1 267.135} C_DIS
LIN {X -0.030,Y -452.517,Z 429.482,A 0.000,B 0.000,C 90.000,E1 266.788} C_DIS
LIN {X 0.160,Y -445.574,Z 429.481,A 0.000,B 0.000,C 90.000,E1 266.502} C_DIS
LIN {X 0.203,Y -437.757,Z 429.479,A 0.000,B 0.000,C 90.000,E1 266.274} C_DIS
LIN {X -0.202,Y -429.617,Z 429.479,A 0.000,B 0.000,C 90.000,E1 266.159} C_DIS
LIN {X 0.178,Y -420.179,Z 429.478,A 0.000,B 0.000,C 90.000,E1 265.988} C_DIS
LIN {X 0.142,Y -410.499,Z 429.478,A 0.000,B 0.000,C 90.000,E1 265.931} C_DIS
LIN {X 0.095,Y -404.370,Z 429.477,A 0.000,B 0.000,C 90.000,E1 265.927} C_DIS
LIN {X 0.010,Y -180.917,Z 429.477,A 0.000,B 0.000,C 90.000,E1 265.927} C_DIS
LIN {X 0.042,Y -180.838,Z 429.472,A 0.000,B 0.000,C 90.000,E1 264.894} C_DIS
LIN {X -0.061,Y -178.879,Z 429.443,A 0.000,B 0.000,C 90.000,E1 259.690} C_DIS
LIN {X 0.015,Y -175.921,Z 429.414,A 0.000,B 0.000,C 90.000,E1 254.574} C_DIS
LIN {X -0.096,Y -174.618,Z 429.405,A 0.000,B 0.000,C 90.000,E1 252.906} C_DIS
LIN {X -0.003,Y -171.599,Z 429.381,A 0.000,B 0.000,C 90.000,E1 248.592} C_DIS
LIN {X -0.014,Y -167.822,Z 429.357,A 0.000,B 0.000,C 90.000,E1 244.280} C_DIS
LIN {X 0.003,Y -166.546,Z 429.347,A 0.000,B 0.000,C 90.000,E1 242.538} C_DIS
LIN {X -0.086,Y -162.542,Z 429.323,A 0.000,B 0.000,C 90.000,E1 238.201} C_DIS
LIN {X -0.025,Y -161.219,Z 429.313,A 0.000,B 0.000,C 90.000,E1 236.421} C_DIS
LIN {X 0.009,Y -157.226,Z 429.289,A 0.000,B 0.000,C 90.000,E1 231.984} C_DIS
LIN {X 0.032,Y -155.952,Z 429.279,A 0.000,B 0.000,C 90.000,E1 230.194} C_DIS
LIN {X -0.009,Y -152.205,Z 429.254,A 0.000,B 0.000,C 90.000,E1 225.729} C_DIS
LIN {X 0.012,Y -150.450,Z 429.239,A 0.000,B 0.000,C 90.000,E1 223.014} C_DIS
LIN {X 0.039,Y -147.176,Z 429.214,A 0.000,B 0.000,C 90.000,E1 218.463} C_DIS
LIN {X 0.005,Y -145.192,Z 429.193,A 0.000,B 0.000,C 90.000,E1 214.818} C_DIS
LIN {X 0.040,Y -142.333,Z 429.163,A 0.000,B 0.000,C 90.000,E1 209.283} C_DIS
LIN {X -0.031,Y -141.723,Z 429.152,A 0.000,B 0.000,C 90.000,E1 207.462} C_DIS
LIN {X -0.048,Y -139.478,Z 429.116,A 0.000,B 0.000,C 90.000,E1 200.972} C_DIS
LIN {X -0.059,Y -138.975,Z 429.101,A 0.000,B 0.000,C 90.000,E1 198.181} C_DIS
LIN {X 0.062,Y -138.332,Z 429.054,A 0.000,B 0.000,C 90.000,E1 189.726} C_DIS
LIN {X 0.065,Y -139.432,Z 429.007,A 0.000,B 0.000,C 90.000,E1 181.318} C_DIS
LIN {X 0.006,Y -140.959,Z 428.976,A 0.000,B 0.000,C 90.000,E1 175.755} C_DIS
LIN {X -0.044,Y -142.715,Z 428.956,A 0.000,B 0.000,C 90.000,E1 172.064} C_DIS
LIN {X 0.055,Y -145.092,Z 428.930,A 0.000,B 0.000,C 90.000,E1 167.409} C_DIS
LIN {X 0.051,Y -147.717,Z 428.910,A 0.000,B 0.000,C 90.000,E1 163.740} C_DIS
LIN {X -0.009,Y -150.375,Z 428.889,A 0.000,B 0.000,C 90.000,E1 160.115} C_DIS
LIN {X 0.010,Y -153.804,Z 428.869,A 0.000,B 0.000,C 90.000,E1 156.485} C_DIS
LIN {X 0.070,Y -157.215,Z 428.849,A 0.000,B 0.000,C 90.000,E1 152.871} C_DIS
LIN {X 0.010,Y -161.381,Z 428.830,A 0.000,B 0.000,C 90.000,E1 149.331} C_DIS
LIN {X 0.021,Y -165.584,Z 428.810,A 0.000,B 0.000,C 90.000,E1 145.801} C_DIS
LIN {X 0.008,Y -170.504,Z 428.791,A 0.000,B 0.000,C 90.000,E1 142.316} C_DIS
LIN {X 0.052,Y -175.384,Z 428.771,A 0.000,B 0.000,C 90.000,E1 138.852} C_DIS
LIN {X -0.085,Y -181.008,Z 428.753,A 0.000,B 0.000,C 90.000,E1 135.486} C_DIS
LIN {X 0.038,Y -186.437,Z 428.734,A 0.000,B 0.000,C 90.000,E1 132.081} C_DIS
LIN {X 0.108,Y -191.062,Z 428.720,A 0.000,B 0.000,C 90.000,E1 129.564} C_DIS
LIN {X 0.012,Y -196.164,Z 428.704,A 0.000,B 0.000,C 90.000,E1 126.664} C_DIS
LIN {X -0.013,Y -294.622,Z 428.704,A 0.000,B 0.000,C 90.000,E1 126.664} C_DIS
LIN {X 0.187,Y -296.871,Z 428.703,A 0.000,B 0.000,C 90.000,E1 126.583} C_DIS
LIN {X 0.046,Y -302.345,Z 428.702,A 0.000,B 0.000,C 90.000,E1 126.297} C_DIS
LIN {X -0.052,Y -305.562,Z 428.700,A 0.000,B 0.000,C 90.000,E1 125.964} C_DIS
LIN {X 0.043,Y -307.551,Z 428.698,A 0.000,B 0.000,C 90.000,E1 125.644} C_DIS
LIN {X -0.044,Y -309.115,Z 428.696,A 0.000,B 0.000,C 90.000,E1 125.358} C_DIS
LIN {X -0.009,Y -310.457,Z 428.695,A 0.000,B 0.000,C 90.000,E1 125.025} C_DIS
LIN {X 0.049,Y -322.386,Z 428.675,A 0.000,B 0.000,C 90.000,E1 121.465} C_DIS
LIN {X 0.067,Y -333.545,Z 428.659,A 0.000,B 0.000,C 90.000,E1 118.615} C_DIS
LIN {X -0.078,Y -346.125,Z 428.644,A 0.000,B 0.000,C 90.000,E1 115.848} C_DIS
LIN {X 0.105,Y -358.589,Z 428.630,A 0.000,B 0.000,C 90.000,E1 113.387} C_DIS
LIN {X -0.150,Y -372.353,Z 428.617,A 0.000,B 0.000,C 90.000,E1 111.046} C_DIS
LIN {X -0.201,Y -387.520,Z 428.604,A 0.000,B 0.000,C 90.000,E1 108.725} C_DIS
LIN {X -0.123,Y -404.199,Z 428.591,A 0.000,B 0.000,C 90.000,E1 106.441} C_DIS
LIN {X 0.160,Y -422.515,Z 428.579,A 0.000,B 0.000,C 90.000,E1 104.189} C_DIS
LIN {X 0.181,Y -442.331,Z 428.567,A 0.000,B 0.000,C 90.000,E1 102.063} C_DIS
LIN {X -0.057,Y -462.790,Z 428.556,A 0.000,B 0.000,C 90.000,E1 100.141} C_DIS
LIN {X 0.208,Y -486.228,Z 428.545,A 0.000,B 0.000,C 90.000,E1 98.106} C_DIS
LIN {X -0.148,Y -488.120,Z 428.544,A 0.000,B 0.000,C 90.000,E1 97.936} C_DIS
LIN {X 0.228,Y -489.798,Z 428.543,A 0.000,B 0.000,C 90.000,E1 97.644} C_DIS
LIN {X 0.118,Y -491.057,Z 428.541,A 0.000,B 0.000,C 90.000,E1 97.409} C_DIS
LIN {X -0.149,Y -492.606,Z 428.539,A 0.000,B 0.000,C 90.000,E1 96.947} C_DIS
LIN {X 0.079,Y -493.092,Z 428.536,A 0.000,B 0.000,C 90.000,E1 96.429} C_DIS
LIN {X -0.173,Y -492.590,Z 428.533,A 0.000,B 0.000,C 90.000,E1 95.967} C_DIS
LIN {X 0.020,Y -491.020,Z 428.530,A 0.000,B 0.000,C 90.000,E1 95.454} C_DIS
LIN {X -0.082,Y -489.747,Z 428.529,A 0.000,B 0.000,C 90.000,E1 95.220} C_DIS
LIN {X 0.144,Y -486.172,Z 428.526,A 0.000,B 0.000,C 90.000,E1 94.702} C_DIS
LIN {X -0.153,Y -476.330,Z 428.519,A 0.000,B 0.000,C 90.000,E1 93.498} C_DIS
LIN {X -0.201,Y -456.791,Z 428.505,A 0.000,B 0.000,C 90.000,E1 90.974} C_DIS
LIN {X -0.097,Y -440.972,Z 428.492,A 0.000,B 0.000,C 90.000,E1 88.625} C_DIS
LIN {X 0.186,Y -424.458,Z 428.478,A 0.000,B 0.000,C 90.000,E1 85.931} C_DIS
LIN {X 0.085,Y -408.800,Z 428.462,A 0.000,B 0.000,C 90.000,E1 83.223} C_DIS
LIN {X -0.105,Y -396.592,Z 428.450,A 0.000,B 0.000,C 90.000,E1 81.027} C_DIS
LIN {X -0.066,Y -384.507,Z 428.438,A 0.000,B 0.000,C 90.000,E1 78.757} C_DIS
LIN {X -0.067,Y -368.367,Z 428.420,A 0.000,B 0.000,C 90.000,E1 75.574} C_DIS
LIN {X -0.013,Y -351.996,Z 428.400,A 0.000,B 0.000,C 90.000,E1 72.000} C_DIS
LIN {X -0.005,Y -339.273,Z 428.383,A 0.000,B 0.000,C 90.000,E1 68.954} C_DIS
LIN {X -0.081,Y -329.496,Z 428.369,A 0.000,B 0.000,C 90.000,E1 66.485} C_DIS
LIN {X -0.060,Y -318.760,Z 428.353,A 0.000,B 0.000,C 90.000,E1 63.640} C_DIS
LIN {X 0.094,Y -308.330,Z 428.337,A 0.000,B 0.000,C 90.000,E1 60.717} C_DIS
LIN {X 0.006,Y -297.291,Z 428.319,A 0.000,B 0.000,C 90.000,E1 57.454} C_DIS
LIN {X 0.010,Y -287.252,Z 428.301,A 0.000,B 0.000,C 90.000,E1 54.116} C_DIS
LIN {X -0.038,Y -279.682,Z 428.286,A 0.000,B 0.000,C 90.000,E1 51.412} C_DIS
LIN {X 0.031,Y -274.011,Z 428.274,A 0.000,B 0.000,C 90.000,E1 49.337} C_DIS
LIN {X 0.145,Y -268.074,Z 428.263,A 0.000,B 0.000,C 90.000,E1 47.229} C_DIS
LIN {X -0.039,Y -261.959,Z 428.251,A 0.000,B 0.000,C 90.000,E1 45.162} C_DIS
LIN {X 0.035,Y -255.692,Z 428.239,A 0.000,B 0.000,C 90.000,E1 43.014} C_DIS
LIN {X 0.007,Y -249.205,Z 428.227,A 0.000,B 0.000,C 90.000,E1 40.862} C_DIS
LIN {X 0.035,Y -240.738,Z 428.211,A 0.000,B 0.000,C 90.000,E1 37.935} C_DIS
LIN {X -0.018,Y -232.803,Z 428.194,A 0.000,B 0.000,C 90.000,E1 34.978} C_DIS
LIN {X -0.006,Y -225.561,Z 428.178,A 0.000,B 0.000,C 90.000,E1 31.957} C_DIS
LIN {X 0.082,Y -219.101,Z 428.161,A 0.000,B 0.000,C 90.000,E1 28.871} C_DIS
LIN {X -0.030,Y -213.323,Z 428.143,A 0.000,B 0.000,C 90.000,E1 25.796} C_DIS
LIN {X 0.038,Y -207.059,Z 428.121,A 0.000,B 0.000,C 90.000,E1 21.844} C_DIS
LIN {X -0.014,Y -201.699,Z 428.099,A 0.000,B 0.000,C 90.000,E1 17.873} C_DIS
LIN {X 0.037,Y -197.356,Z 428.077,A 0.000,B 0.000,C 90.000,E1 13.828} C_DIS
LIN {X -0.064,Y -193.340,Z 428.050,A 0.000,B 0.000,C 90.000,E1 8.973} C_DIS
LIN {X -0.022,Y -190.500,Z 428.018,A 0.000,B 0.000,C 90.000,E1 3.212} C_DIS
LIN {X 0.026,Y -190.535,Z 427.965,A 0.000,B 0.000,C 90.000,E1 353.742} C_DIS
LIN {X -0.024,Y -193.314,Z 427.933,A 0.000,B 0.000,C 90.000,E1 347.993} C_DIS
LIN {X -0.029,Y -197.142,Z 427.906,A 0.000,B 0.000,C 90.000,E1 343.087} C_DIS
LIN {X -0.020,Y -201.406,Z 427.883,A 0.000,B 0.000,C 90.000,E1 339.028} C_DIS
LIN {X 0.122,Y -206.766,Z 427.861,A 0.000,B 0.000,C 90.000,E1 334.973} C_DIS
LIN {X -0.046,Y -213.010,Z 427.839,A 0.000,B 0.000,C 90.000,E1 331.051} C_DIS
LIN {X 0.019,Y -219.828,Z 427.817,A 0.000,B 0.000,C 90.000,E1 327.120} C_DIS
LIN {X 0.048,Y -227.240,Z 427.796,A 0.000,B 0.000,C 90.000,E1 323.256} C_DIS
LIN {X -0.019,Y -233.867,Z 427.779,A 0.000,B 0.000,C 90.000,E1 320.231} C_DIS
LIN {X -0.012,Y -241.175,Z 427.762,A 0.000,B 0.000,C 90.000,E1 317.229} C_DIS
LIN {X -0.166,Y -250.345,Z 427.744,A 0.000,B 0.000,C 90.000,E1 313.947} C_DIS
LIN {X -0.035,Y -260.864,Z 427.726,A 0.000,B 0.000,C 90.000,E1 310.663} C_DIS
LIN {X 0.136,Y -272.519,Z 427.708,A 0.000,B 0.000,C 90.000,E1 307.443} C_DIS
LIN {X 0.160,Y -285.038,Z 427.691,A 0.000,B 0.000,C 90.000,E1 304.326} C_DIS
LIN {X -0.093,Y -295.118,Z 427.678,A 0.000,B 0.000,C 90.000,E1 302.005} C_DIS
LIN {X 0.023,Y -309.048,Z 427.661,A 0.000,B 0.000,C 90.000,E1 298.999} C_DIS
LIN {X -0.054,Y -320.667,Z 427.649,A 0.000,B 0.000,C 90.000,E1 296.744} C_DIS
LIN {X -0.078,Y -336.908,Z 427.633,A 0.000,B 0.000,C 90.000,E1 293.898} C_DIS
LIN {X 0.199,Y -359.753,Z 427.614,A 0.000,B 0.000,C 90.000,E1 290.482} C_DIS
LIN {X -0.156,Y -380.429,Z 427.599,A 0.000,B 0.000,C 90.000,E1 287.873} C_DIS
LIN {X 0.014,Y -395.147,Z 427.590,A 0.000,B 0.000,C 90.000,E1 286.134} C_DIS
LIN {X -0.096,Y -407.772,Z 427.582,A 0.000,B 0.000,C 90.000,E1 284.828} C_DIS
LIN {X -0.185,Y -425.984,Z 427.572,A 0.000,B 0.000,C 90.000,E1 283.063} C_DIS
LIN {X -0.121,Y -433.653,Z 427.568,A 0.000,B 0.000,C 90.000,E1 282.299} C_DIS
LIN {X -0.184,Y -441.083,Z 427.564,A 0.000,B 0.000,C 90.000,E1 281.535} C_DIS
LIN {X -0.172,Y -450.521,Z 427.558,A 0.000,B 0.000,C 90.000,E1 280.489} C_DIS
LIN {X 0.133,Y -457.023,Z 427.554,A 0.000,B 0.000,C 90.000,E1 279.670} C_DIS
LIN {X 0.248,Y -464.875,Z 427.548,A 0.000,B 0.000,C 90.000,E1 278.624} C_DIS
LIN {X -0.074,Y -471.776,Z 427.542,A 0.000,B 0.000,C 90.000,E1 277.644} C_DIS
LIN {X 0.155,Y -478.107,Z 427.537,A 0.000,B 0.000,C 90.000,E1 276.606} C_DIS
LIN {X 0.163,Y -482.330,Z 427.533,A 0.000,B 0.000,C 90.000,E1 275.853} C_DIS
LIN {X 0.160,Y -485.912,Z 427.528,A 0.000,B 0.000,C 90.000,E1 275.106} C_DIS
LIN {X -0.011,Y -486.959,Z 427.527,A 0.000,B 0.000,C 90.000,E1 274.878} C_DIS
LIN {X 0.188,Y -488.704,Z 427.524,A 0.000,B 0.000,C 90.000,E1 274.359} C_DIS
LIN {X -0.099,Y -490.058,Z 427.522,A 0.000,B 0.000,C 90.000,E1 273.898} C_DIS
LIN {X 0.081,Y -491.110,Z 427.519,A 0.000,B 0.000,C 90.000,E1 273.383} C_DIS
LIN {X -0.192,Y -491.818,Z 427.516,A 0.000,B 0.000,C 90.000,E1 272.922} C_DIS
LIN {X 0.006,Y -492.156,Z 427.513,A 0.000,B 0.000,C 90.000,E1 272.407} C_DIS
LIN {X 0.211,Y -492.104,Z 427.511,A 0.000,B 0.000,C 90.000,E1 271.892} C_DIS
LIN {X -0.059,Y -491.640,Z 427.508,A 0.000,B 0.000,C 90.000,E1 271.432} C_DIS
LIN {X 0.148,Y -490.712,Z 427.505,A 0.000,B 0.000,C 90.000,E1 270.917} C_DIS
LIN {X -0.138,Y -489.258,Z 427.502,A 0.000,B 0.000,C 90.000,E1 270.458} C_DIS
LIN {X 0.062,Y -487.309,Z 427.500,A 0.000,B 0.000,C 90.000,E1 269.943} C_DIS
LIN {X -0.233,Y -484.757,Z 427.497,A 0.000,B 0.000,C 90.000,E1 269.484} C_DIS
LIN {X -0.061,Y -481.553,Z 427.494,A 0.000,B 0.000,C 90.000,E1 268.969} C_DIS
LIN {X 0.090,Y -477.403,Z 427.491,A 0.000,B 0.000,C 90.000,E1 268.453} C_DIS
LIN {X -0.083,Y -475.027,Z 427.490,A 0.000,B 0.000,C 90.000,E1 268.224} C_DIS
LIN {X 0.196,Y -469.450,Z 427.487,A 0.000,B 0.000,C 90.000,E1 267.707} C_DIS
LIN {X 0.159,Y -466.205,Z 427.486,A 0.000,B 0.000,C 90.000,E1 267.478} C_DIS
LIN {X 0.187,Y -459.545,Z 427.484,A 0.000,B 0.000,C 90.000,E1 267.078} C_DIS
LIN {X -0.142,Y -452.342,Z 427.482,A 0.000,B 0.000,C 90.000,E1 266.788} C_DIS
LIN {X 0.048,Y -445.216,Z 427.481,A 0.000,B 0.000,C 90.000,E1 266.502} C_DIS
LIN {X 0.121,Y -437.367,Z 427.479,A 0.000,B 0.000,C 90.000,E1 266.274} C_DIS
LIN {X 0.201,Y -429.423,Z 427.478,A 0.000,B 0.000,C 90.000,E1 266.102} C_DIS
LIN {X 0.174,Y -420.250,Z 427.478,A 0.000,B 0.000,C 90.000,E1 265.988} C_DIS
LIN {X 0.138,Y -410.452,Z 427.478,A 0.000,B 0.000,C 90.000,E1 265.931} C_DIS
LIN {X 0.041,Y -180.918,Z 427.477,A 0.000,B 0.000,C 90.000,E1 265.927} C_DIS
LIN {X 0.072,Y -180.840,Z 427.472,A 0.000,B 0.000,C 90.000,E1 264.894} C_DIS
LIN {X -0.031,Y -178.883,Z 427.443,A 0.000,B 0.000,C 90.000,E1 259.690} C_DIS
LIN {X 0.043,Y -175.925,Z 427.414,A 0.000,B 0.000,C 90.000,E1 254.574} C_DIS
LIN {X -0.010,Y -175.364,Z 427.410,A 0.000,B 0.000,C 90.000,E1 253.740} C_DIS
LIN {X 0.048,Y -172.142,Z 427.386,A 0.000,B 0.000,C 90.000,E1 249.444} C_DIS
LIN {X 0.026,Y -171.606,Z 427.381,A 0.000,B 0.000,C 90.000,E1 248.592} C_DIS
LIN {X 0.013,Y -167.829,Z 427.357,A 0.000,B 0.000,C 90.000,E1 244.280} C_DIS
LIN {X 0.031,Y -166.555,Z 427.348,A 0.000,B 0.000,C 90.000,E1 242.538} C_DIS
LIN {X -0.059,Y -162.550,Z 427.323,A 0.000,B 0.000,C 90.000,E1 238.201} C_DIS
LIN {X 0.002,Y -161.228,Z 427.313,A 0.000,B 0.000,C 90.000,E1 236.421} C_DIS
LIN {X 0.036,Y -157.234,Z 427.289,A 0.000,B 0.000,C 90.000,E1 231.984} C_DIS
LIN {X 0.059,Y -155.958,Z 427.279,A 0.000,B 0.000,C 90.000,E1 230.194} C_DIS
LIN {X 0.018,Y -152.212,Z 427.254,A 0.000,B 0.000,C 90.000,E1 225.729} C_DIS
LIN {X 0.038,Y -150.457,Z 427.239,A 0.000,B 0.000,C 90.000,E1 223.014} C_DIS
LIN {X 0.065,Y -147.182,Z 427.214,A 0.000,B 0.000,C 90.000,E1 218.463} C_DIS
LIN {X 0.031,Y -145.199,Z 427.194,A 0.000,B 0.000,C 90.000,E1 214.818} C_DIS
LIN {X -0.059,Y -142.337,Z 427.163,A 0.000,B 0.000,C 90.000,E1 209.333} C_DIS
LIN {X -0.005,Y -141.726,Z 427.153,A 0.000,B 0.000,C 90.000,E1 207.462} C_DIS
LIN {X -0.023,Y -139.479,Z 427.116,A 0.000,B 0.000,C 90.000,E1 200.972} C_DIS
LIN {X -0.034,Y -138.978,Z 427.101,A 0.000,B 0.000,C 90.000,E1 198.181} C_DIS
LIN {X -0.049,Y -138.332,Z 427.054,A 0.000,B 0.000,C 90.000,E1 189.782} C_DIS
LIN {X -0.049,Y -139.430,Z 427.008,A 0.000,B 0.000,C 90.000,E1 181.375} C_DIS
LIN {X 0.005,Y -141.358,Z 426.971,A 0.000,B 0.000,C 90.000,E1 174.837} C_DIS
LIN {X -0.019,Y -142.711,Z 426.956,A 0.000,B 0.000,C 90.000,E1 172.064} C_DIS
LIN {X -0.060,Y -145.086,Z 426.930,A 0.000,B 0.000,C 90.000,E1 167.465} C_DIS
LIN {X 0.077,Y -147.711,Z 426.910,A 0.000,B 0.000,C 90.000,E1 163.740} C_DIS
LIN {X 0.018,Y -150.366,Z 426.890,A 0.000,B 0.000,C 90.000,E1 160.115} C_DIS
LIN {X 0.037,Y -153.793,Z 426.869,A 0.000,B 0.000,C 90.000,E1 156.485} C_DIS
LIN {X -0.043,Y -157.205,Z 426.849,A 0.000,B 0.000,C 90.000,E1 152.922} C_DIS
LIN {X 0.038,Y -161.368,Z 426.830,A 0.000,B 0.000,C 90.000,E1 149.331} C_DIS
LIN {X 0.050,Y -165.570,Z 426.810,A 0.000,B 0.000,C 90.000,E1 145.801} C_DIS
LIN {X -0.067,Y -170.489,Z 426.791,A 0.000,B 0.000,C 90.000,E1 142.351} C_DIS
LIN {X 0.082,Y -175.370,Z 426.772,A 0.000,B 0.000,C 90.000,E1 138.852} C_DIS
LIN {X -0.055,Y -180.994,Z 426.753,A 0.000,B 0.000,C 90.000,E1 135.486} C_DIS
LIN {X 0.069,Y -186.421,Z 426.734,A 0.000,B 0.000,C 90.000,E1 132.081} C_DIS
LIN {X 0.017,Y -191.048,Z 426.720,A 0.000,B 0.000,C 90.000,E1 129.600} C_DIS
LIN {X 0.114,Y -196.259,Z 426.703,A 0.000,B 0.000,C 90.000,E1 126.583} C_DIS
LIN {X 0.118,Y -295.277,Z 426.703,A 0.000,B 0.000,C 90.000,E1 126.583} C_DIS
LIN {X 0.012,Y -296.416,Z 426.703,A 0.000,B 0.000,C 90.000,E1 126.583} C_DIS
LIN {X 0.094,Y -301.776,Z 426.702,A 0.000,B 0.000,C 90.000,E1 126.297} C_DIS
LIN {X -0.044,Y -304.930,Z 426.700,A 0.000,B 0.000,C 90.000,E1 126.011} C_DIS
LIN {X 0.015,Y -308.566,Z 426.697,A 0.000,B 0.000,C 90.000,E1 125.438} C_DIS
LIN {X 0.043,Y -310.057,Z 426.695,A 0.000,B 0.000,C 90.000,E1 125.105} C_DIS
LIN {X 0.085,Y -313.275,Z 426.690,A 0.000,B 0.000,C 90.000,E1 124.119} C_DIS
LIN {X -0.100,Y -323.220,Z 426.674,A 0.000,B 0.000,C 90.000,E1 121.258} C_DIS
LIN {X -0.070,Y -334.492,Z 426.658,A 0.000,B 0.000,C 90.000,E1 118.409} C_DIS
LIN {X 0.116,Y -347.188,Z 426.642,A 0.000,B 0.000,C 90.000,E1 115.591} C_DIS
LIN {X -0.140,Y -359.766,Z 426.629,A 0.000,B 0.000,C 90.000,E1 113.206} C_DIS
LIN {X 0.111,Y -373.655,Z 426.616,A 0.000,B 0.000,C 90.000,E1 110.791} C_DIS
LIN {X -0.028,Y -388.954,Z 426.603,A 0.000,B 0.000,C 90.000,E1 108.489} C_DIS
LIN {X 0.099,Y -405.777,Z 426.590,A 0.000,B 0.000,C 90.000,E1 106.205} C_DIS
LIN {X 0.023,Y -424.248,Z 426.578,A 0.000,B 0.000,C 90.000,E1 104.008} C_DIS
LIN {X 0.141,Y -444.146,Z 426.566,A 0.000,B 0.000,C 90.000,E1 101.883} C_DIS
LIN {X 0.018,Y -464.653,Z 426.555,A 0.000,B 0.000,C 90.000,E1 99.962} C_DIS
LIN {X 0.203,Y -485.623,Z 426.545,A 0.000,B 0.000,C 90.000,E1 98.163} C_DIS
LIN {X -0.159,Y -487.710,Z 426.544,A 0.000,B 0.000,C 90.000,E1 97.992} C_DIS
LIN {X 0.225,Y -489.533,Z 426.543,A 0.000,B 0.000,C 90.000,E1 97.701} C_DIS
LIN {X 0.059,Y -490.903,Z 426.542,A 0.000,B 0.000,C 90.000,E1 97.473} C_DIS
LIN {X -0.146,Y -492.631,Z 426.539,A 0.000,B 0.000,C 90.000,E1 97.004} C_DIS
LIN {X 0.081,Y -493.265,Z 426.536,A 0.000,B 0.000,C 90.000,E1 96.486} C_DIS
LIN {X -0.171,Y -492.911,Z 426.533,A 0.000,B 0.000,C 90.000,E1 96.024} C_DIS
LIN {X 0.022,Y -491.512,Z 426.531,A 0.000,B 0.000,C 90.000,E1 95.511} C_DIS
LIN {X -0.080,Y -490.348,Z 426.529,A 0.000,B 0.000,C 90.000,E1 95.277} C_DIS
LIN {X -0.226,Y -488.787,Z 426.528,A 0.000,B 0.000,C 90.000,E1 95.049} C_DIS
LIN {X 0.195,Y -481.080,Z 426.522,A 0.000,B 0.000,C 90.000,E1 94.012} C_DIS
LIN {X 0.188,Y -465.178,Z 426.511,A 0.000,B 0.000,C 90.000,E1 92.007} C_DIS
LIN {X -0.159,Y -450.255,Z 426.500,A 0.000,B 0.000,C 90.000,E1 90.000} C_DIS
LIN {X 0.106,Y -431.595,Z 426.484,A 0.000,B 0.000,C 90.000,E1 87.078} C_DIS
LIN {X -0.149,Y -414.025,Z 426.467,A 0.000,B 0.000,C 90.000,E1 84.147} C_DIS
LIN {X 0.187,Y -401.729,Z 426.455,A 0.000,B 0.000,C 90.000,E1 81.894} C_DIS
LIN {X -0.107,Y -389.592,Z 426.443,A 0.000,B 0.000,C 90.000,E1 79.690} C_DIS
LIN {X -0.185,Y -379.075,Z 426.432,A 0.000,B 0.000,C 90.000,E1 77.701} C_DIS
LIN {X 0.040,Y -366.109,Z 426.417,A 0.000,B 0.000,C 90.000,E1 75.046} C_DIS
LIN {X 0.105,Y -349.898,Z 426.397,A 0.000,B 0.000,C 90.000,E1 71.456} C_DIS
LIN {X 0.044,Y -337.276,Z 426.380,A 0.000,B 0.000,C 90.000,E1 68.411} C_DIS
LIN {X 0.042,Y -327.513,Z 426.366,A 0.000,B 0.000,C 90.000,E1 65.921} C_DIS
LIN {X 0.001,Y -316.811,Z 426.350,A 0.000,B 0.000,C 90.000,E1 63.076} C_DIS
LIN {X -0.139,Y -305.294,Z 426.332,A 0.000,B 0.000,C 90.000,E1 59.871} C_DIS
LIN {X 0.017,Y -293.471,Z 426.312,A 0.000,B 0.000,C 90.000,E1 56.215} C_DIS
LIN {X 0.069,Y -283.705,Z 426.294,A 0.000,B 0.000,C 90.000,E1 52.844} C_DIS
LIN {X 0.058,Y -276.181,Z 426.278,A 0.000,B 0.000,C 90.000,E1 50.114} C_DIS
LIN {X -0.140,Y -270.374,Z 426.267,A 0.000,B 0.000,C 90.000,E1 48.081} C_DIS
LIN {X -0.086,Y -264.332,Z 426.255,A 0.000,B 0.000,C 90.000,E1 45.972} C_DIS
LIN {X -0.152,Y -258.139,Z 426.243,A 0.000,B 0.000,C 90.000,E1 43.866} C_DIS
LIN {X 0.036,Y -251.755,Z 426.232,A 0.000,B 0.000,C 90.000,E1 41.676} C_DIS
LIN {X 0.125,Y -243.175,Z 426.215,A 0.000,B 0.000,C 90.000,E1 38.749} C_DIS
LIN {X 0.078,Y -235.041,Z 426.199,A 0.000,B 0.000,C 90.000,E1 35.804} C_DIS
LIN {X -0.051,Y -227.627,Z 426.182,A 0.000,B 0.000,C 90.000,E1 32.832} C_DIS
LIN {X 0.091,Y -220.950,Z 426.165,A 0.000,B 0.000,C 90.000,E1 29.745} C_DIS
LIN {X 0.032,Y -214.963,Z 426.148,A 0.000,B 0.000,C 90.000,E1 26.668} C_DIS
LIN {X 0.110,Y -209.652,Z 426.131,A 0.000,B 0.000,C 90.000,E1 23.515} C_DIS
LIN {X 0.016,Y -203.890,Z 426.109,A 0.000,B 0.000,C 90.000,E1 19.577} C_DIS
LIN {X 0.060,Y -199.054,Z 426.086,A 0.000,B 0.000,C 90.000,E1 15.552} C_DIS
LIN {X -0.045,Y -194.572,Z 426.059,A 0.000,B 0.000,C 90.000,E1 10.715} C_DIS
LIN {X -0.026,Y -191.477,Z 426.032,A 0.000,B 0.000,C 90.000,E1 5.796} C_DIS
LIN {X 0.000,Y -189.716,Z 425.988,A 0.000,B 0.000,C 90.000,E1 357.879} C_DIS
LIN {X 0.024,Y -191.799,Z 425.947,A 0.000,B 0.000,C 90.000,E1 350.443} C_DIS
LIN {X 0.018,Y -194.932,Z 425.920,A 0.000,B 0.000,C 90.000,E1 345.519} C_DIS
LIN {X -0.031,Y -198.597,Z 425.897,A 0.000,B 0.000,C 90.000,E1 341.456} C_DIS
LIN {X -0.020,Y -203.282,Z 425.874,A 0.000,B 0.000,C 90.000,E1 337.411} C_DIS
LIN {X 0.083,Y -209.009,Z 425.852,A 0.000,B 0.000,C 90.000,E1 333.384} C_DIS
LIN {X -0.001,Y -215.551,Z 425.830,A 0.000,B 0.000,C 90.000,E1 329.459} C_DIS
LIN {X -0.112,Y -222.592,Z 425.809,A 0.000,B 0.000,C 90.000,E1 325.595} C_DIS
LIN {X -0.044,Y -230.324,Z 425.787,A 0.000,B 0.000,C 90.000,E1 321.743} C_DIS
LIN {X 0.014,Y -239.160,Z 425.766,A 0.000,B 0.000,C 90.000,E1 317.957} C_DIS
LIN {X -0.033,Y -248.111,Z 425.748,A 0.000,B 0.000,C 90.000,E1 314.636} C_DIS
LIN {X -0.002,Y -255.947,Z 425.734,A 0.000,B 0.000,C 90.000,E1 312.081} C_DIS
LIN {X 0.163,Y -267.107,Z 425.716,A 0.000,B 0.000,C 90.000,E1 308.830} C_DIS
LIN {X -0.123,Y -277.873,Z 425.700,A 0.000,B 0.000,C 90.000,E1 306.091} C_DIS
LIN {X 0.151,Y -289.317,Z 425.685,A 0.000,B 0.000,C 90.000,E1 303.293} C_DIS
LIN {X -0.162,Y -301.131,Z 425.670,A 0.000,B 0.000,C 90.000,E1 300.669} C_DIS
LIN {X -0.029,Y -315.515,Z 425.654,A 0.000,B 0.000,C 90.000,E1 297.692} C_DIS
LIN {X -0.105,Y -333.149,Z 425.636,A 0.000,B 0.000,C 90.000,E1 294.515} C_DIS
LIN {X -0.067,Y -342.964,Z 425.627,A 0.000,B 0.000,C 90.000,E1 292.950} C_DIS
LIN {X 0.033,Y -362.080,Z 425.612,A 0.000,B 0.000,C 90.000,E1 290.194} C_DIS
LIN {X 0.009,Y -378.207,Z 425.601,A 0.000,B 0.000,C 90.000,E1 288.127} C_DIS
LIN {X 0.191,Y -390.107,Z 425.593,A 0.000,B 0.000,C 90.000,E1 286.677} C_DIS
LIN {X 0.058,Y -402.791,Z 425.585,A 0.000,B 0.000,C 90.000,E1 285.315} C_DIS
LIN {X -0.102,Y -421.044,Z 425.575,A 0.000,B 0.000,C 90.000,E1 283.536} C_DIS
LIN {X -0.141,Y -431.389,Z 425.570,A 0.000,B 0.000,C 90.000,E1 282.535} C_DIS
LIN {X -0.157,Y -441.097,Z 425.564,A 0.000,B 0.000,C 90.000,E1 281.535} C_DIS
LIN {X 0.071,Y -448.344,Z 425.560,A 0.000,B 0.000,C 90.000,E1 280.715} C_DIS
LIN {X -0.178,Y -455.011,Z 425.555,A 0.000,B 0.000,C 90.000,E1 279.962} C_DIS
LIN {X -0.090,Y -463.066,Z 425.549,A 0.000,B 0.000,C 90.000,E1 278.916} C_DIS
LIN {X 0.093,Y -470.135,Z 425.544,A 0.000,B 0.000,C 90.000,E1 277.871} C_DIS
LIN {X -0.173,Y -476.647,Z 425.538,A 0.000,B 0.000,C 90.000,E1 276.891} C_DIS
LIN {X -0.230,Y -481.029,Z 425.534,A 0.000,B 0.000,C 90.000,E1 276.144} C_DIS
LIN {X -0.203,Y -484.832,Z 425.530,A 0.000,B 0.000,C 90.000,E1 275.391} C_DIS
LIN {X -0.063,Y -486.961,Z 425.527,A 0.000,B 0.000,C 90.000,E1 274.878} C_DIS
LIN {X 0.136,Y -488.679,Z 425.524,A 0.000,B 0.000,C 90.000,E1 274.359} C_DIS
LIN {X -0.151,Y -490.043,Z 425.522,A 0.000,B 0.000,C 90.000,E1 273.898} C_DIS
LIN {X 0.029,Y -491.118,Z 425.519,A 0.000,B 0.000,C 90.000,E1 273.383} C_DIS
LIN {X 0.247,Y -491.835,Z 425.516,A 0.000,B 0.000,C 90.000,E1 272.865} C_DIS
LIN {X -0.047,Y -492.196,Z 425.513,A 0.000,B 0.000,C 90.000,E1 272.407} C_DIS
LIN {X 0.159,Y -492.112,Z 425.511,A 0.000,B 0.000,C 90.000,E1 271.892} C_DIS
LIN {X -0.111,Y -491.640,Z 425.508,A 0.000,B 0.000,C 90.000,E1 271.432} C_DIS
LIN {X 0.095,Y -490.727,Z 425.505,A 0.000,B 0.000,C 90.000,E1 270.917} C_DIS
LIN {X -0.189,Y -489.297,Z 425.502,A 0.000,B 0.000,C 90.000,E1 270.458} C_DIS
LIN {X 0.010,Y -487.360,Z 425.500,A 0.000,B 0.000,C 90.000,E1 269.943} C_DIS
LIN {X 0.200,Y -484.801,Z 425.497,A 0.000,B 0.000,C 90.000,E1 269.427} C_DIS
LIN {X -0.113,Y -481.582,Z 425.494,A 0.000,B 0.000,C 90.000,E1 268.969} C_DIS
LIN {X 0.040,Y -477.455,Z 425.491,A 0.000,B 0.000,C 90.000,E1 268.453} C_DIS
LIN {X 0.183,Y -472.307,Z 425.489,A 0.000,B 0.000,C 90.000,E1 267.936} C_DIS
LIN {X 0.136,Y -469.457,Z 425.487,A 0.000,B 0.000,C 90.000,E1 267.707} C_DIS
LIN {X 0.089,Y -466.181,Z 425.486,A 0.000,B 0.000,C 90.000,E1 267.478} C_DIS
LIN {X -0.123,Y -463.060,Z 425.485,A 0.000,B 0.000,C 90.000,E1 267.306} C_DIS
LIN {X 0.203,Y -456.221,Z 425.483,A 0.000,B 0.000,C 90.000,E1 266.906} C_DIS
LIN {X 0.179,Y -449.152,Z 425.481,A 0.000,B 0.000,C 90.000,E1 266.617} C_DIS
LIN {X 0.132,Y -441.926,Z 425.480,A 0.000,B 0.000,C 90.000,E1 266.388} C_DIS
LIN {X 0.016,Y -434.341,Z 425.479,A 0.000,B 0.000,C 90.000,E1 266.216} C_DIS
LIN {X -0.187,Y -426.101,Z 425.478,A 0.000,B 0.000,C 90.000,E1 266.102} C_DIS
LIN {X -0.094,Y -415.327,Z 425.478,A 0.000,B 0.000,C 90.000,E1 265.988} C_DIS
LIN {X 0.116,Y -407.768,Z 425.477,A 0.000,B 0.000,C 90.000,E1 265.927} C_DIS
LIN {X 0.018,Y -180.918,Z 425.477,A 0.000,B 0.000,C 90.000,E1 265.927} C_DIS
LIN {X 0.048,Y -180.838,Z 425.472,A 0.000,B 0.000,C 90.000,E1 264.894} C_DIS
LIN {X -0.054,Y -178.880,Z 425.443,A 0.000,B 0.000,C 90.000,E1 259.690} C_DIS
LIN {X 0.022,Y -175.922,Z 425.414,A 0.000,B 0.000,C 90.000,E1 254.574} C_DIS
LIN {X -0.089,Y -174.621,Z 425.405,A 0.000,B 0.000,C 90.000,E1 252.906} C_DIS
LIN {X 0.003,Y -171.601,Z 425.381,A 0.000,B 0.000,C 90.000,E1 248.592} C_DIS
LIN {X -0.008,Y -167.824,Z 425.357,A 0.000,B 0.000,C 90.000,E1 244.280} C_DIS
LIN {X 0.009,Y -166.548,Z 425.347,A 0.000,B 0.000,C 90.000,E1 242.538} C_DIS
LIN {X -0.080,Y -162.545,Z 425.323,A 0.000,B 0.000,C 90.000,E1 238.201} C_DIS
LIN {X -0.019,Y -161.221,Z 425.313,A 0.000,B 0.000,C 90.000,E1 236.421} C_DIS
LIN {X 0.015,Y -157.228,Z 425.289,A 0.000,B 0.000,C 90.000,E1 231.984} C_DIS
LIN {X 0.039,Y -155.953,Z 425.279,A 0.000,B 0.000,C 90.000,E1 230.194} C_DIS
LIN {X -0.003,Y -152.206,Z 425.254,A 0.000,B 0.000,C 90.000,E1 225.729} C_DIS
LIN {X 0.018,Y -150.452,Z 425.239,A 0.000,B 0.000,C 90.000,E1 223.014} C_DIS
LIN {X 0.045,Y -147.177,Z 425.214,A 0.000,B 0.000,C 90.000,E1 218.463} C_DIS
LIN {X 0.012,Y -145.194,Z 425.193,A 0.000,B 0.000,C 90.000,E1 214.818} C_DIS
LIN {X 0.046,Y -142.335,Z 425.163,A 0.000,B 0.000,C 90.000,E1 209.283} C_DIS
LIN {X -0.025,Y -141.724,Z 425.153,A 0.000,B 0.000,C 90.000,E1 207.462} C_DIS
LIN {X -0.042,Y -139.478,Z 425.116,A 0.000,B 0.000,C 90.000,E1 200.972} C_DIS
LIN {X -0.054,Y -138.976,Z 425.101,A 0.000,B 0.000,C 90.000,E1 198.181} C_DIS
LIN {X 0.068,Y -138.332,Z 425.054,A 0.000,B 0.000,C 90.000,E1 189.726} C_DIS
LIN {X -0.068,Y -139.431,Z 425.007,A 0.000,B 0.000,C 90.000,E1 181.375} C_DIS
LIN {X 0.012,Y -140.958,Z 424.976,A 0.000,B 0.000,C 90.000,E1 175.755} C_DIS
LIN {X -0.038,Y -142.714,Z 424.956,A 0.000,B 0.000,C 90.000,E1 172.064} C_DIS
LIN {X 0.061,Y -145.091,Z 424.930,A 0.000,B 0.000,C 90.000,E1 167.409} C_DIS
LIN {X 0.057,Y -147.716,Z 424.910,A 0.000,B 0.000,C 90.000,E1 163.740} C_DIS
LIN {X -0.002,Y -150.372,Z 424.890,A 0.000,B 0.000,C 90.000,E1 160.115} C_DIS
LIN {X 0.015,Y -153.802,Z 424.869,A 0.000,B 0.000,C 90.000,E1 156.485} C_DIS
LIN {X 0.075,Y -157.214,Z 424.849,A 0.000,B 0.000,C 90.000,E1 152.871} C_DIS
LIN {X 0.016,Y -161.378,Z 424.830,A 0.000,B 0.000,C 90.000,E1 149.331} C_DIS
LIN {X 0.028,Y -165.580,Z 424.810,A 0.000,B 0.000,C 90.000,E1 145.801} C_DIS
LIN {X 0.015,Y -170.500,Z 424.791,A 0.000,B 0.000,C 90.000,E1 142.316} C_DIS
LIN {X 0.059,Y -175.381,Z 424.772,A 0.000,B 0.000,C 90.000,E1 138.852} C_DIS
LIN {X -0.079,Y -181.005,Z 424.753,A 0.000,B 0.000,C 90.000,E1 135.486} C_DIS
LIN {X 0.046,Y -186.434,Z 424.734,A 0.000,B 0.000,C 90.000,E1 132.081} C_DIS
LIN {X 0.115,Y -191.060,Z 424.720,A 0.000,B 0.000,C 90.000,E1 129.564} C_DIS
LIN {X -0.052,Y -196.350,Z 424.703,A 0.000,B 0.000,C 90.000,E1 126.583} C_DIS
LIN {X -0.124,Y -295.211,Z 424.703,A 0.000,B 0.000,C 90.000,E1 126.583} C_DIS
LIN {X 0.021,Y -296.323,Z 424.703,A 0.000,B 0.000,C 90.000,E1 126.537} C_DIS
LIN {X 0.057,Y -301.348,Z 424.702,A 0.000,B 0.000,C 90.000,E1 126.297} C_DIS
LIN {X 0.044,Y -304.495,Z 424.700,A 0.000,B 0.000,C 90.000,E1 126.011} C_DIS
LIN {X -0.148,Y -308.172,Z 424.697,A 0.000,B 0.000,C 90.000,E1 125.518} C_DIS
LIN {X 0.056,Y -309.777,Z 424.695,A 0.000,B 0.000,C 90.000,E1 125.152} C_DIS
LIN {X -0.129,Y -312.073,Z 424.692,A 0.000,B 0.000,C 90.000,E1 124.532} C_DIS
LIN {X 0.084,Y -321.857,Z 424.676,A 0.000,B 0.000,C 90.000,E1 121.592} C_DIS
LIN {X 0.085,Y -332.951,Z 424.660,A 0.000,B 0.000,C 90.000,E1 118.743} C_DIS
LIN {X -0.077,Y -345.463,Z 424.644,A 0.000,B 0.000,C 90.000,E1 115.976} C_DIS
LIN {X 0.089,Y -357.861,Z 424.631,A 0.000,B 0.000,C 90.000,E1 113.515} C_DIS
LIN {X -0.048,Y -371.554,Z 424.617,A 0.000,B 0.000,C 90.000,E1 111.153} C_DIS
LIN {X -0.125,Y -386.645,Z 424.605,A 0.000,B 0.000,C 90.000,E1 108.833} C_DIS
LIN {X -0.077,Y -403.242,Z 424.592,A 0.000,B 0.000,C 90.000,E1 106.551} C_DIS
LIN {X 0.175,Y -421.469,Z 424.580,A 0.000,B 0.000,C 90.000,E1 104.300} C_DIS
LIN {X 0.036,Y -441.236,Z 424.568,A 0.000,B 0.000,C 90.000,E1 102.187} C_DIS
LIN {X -0.191,Y -461.665,Z 424.557,A 0.000,B 0.000,C 90.000,E1 100.254} C_DIS
LIN {X -0.015,Y -485.241,Z 424.546,A 0.000,B 0.000,C 90.000,E1 98.219} C_DIS
LIN {X 0.103,Y -487.471,Z 424.544,A 0.000,B 0.000,C 90.000,E1 97.992} C_DIS
LIN {X 0.081,Y -489.337,Z 424.543,A 0.000,B 0.000,C 90.000,E1 97.757} C_DIS
LIN {X -0.006,Y -490.753,Z 424.542,A 0.000,B 0.000,C 90.000,E1 97.530} C_DIS
LIN {X 0.216,Y -492.644,Z 424.539,A 0.000,B 0.000,C 90.000,E1 97.011} C_DIS
LIN {X -0.042,Y -493.414,Z 424.536,A 0.000,B 0.000,C 90.000,E1 96.549} C_DIS
LIN {X 0.199,Y -493.195,Z 424.534,A 0.000,B 0.000,C 90.000,E1 96.030} C_DIS
LIN {X -0.047,Y -491.948,Z 424.531,A 0.000,B 0.000,C 90.000,E1 95.568} C_DIS
LIN {X -0.147,Y -490.875,Z 424.530,A 0.000,B 0.000,C 90.000,E1 95.334} C_DIS
LIN {X 0.196,Y -489.430,Z 424.528,A 0.000,B 0.000,C 90.000,E1 95.049} C_DIS
LIN {X 0.103,Y -481.809,Z 424.523,A 0.000,B 0.000,C 90.000,E1 94.073} C_DIS
LIN {X 0.145,Y -465.883,Z 424.512,A 0.000,B 0.000,C 90.000,E1 92.064} C_DIS
LIN {X -0.185,Y -450.896,Z 424.500,A 0.000,B 0.000,C 90.000,E1 90.057} C_DIS
LIN {X 0.101,Y -432.167,Z 424.484,A 0.000,B 0.000,C 90.000,E1 87.135} C_DIS
LIN {X -0.008,Y -413.026,Z 424.466,A 0.000,B 0.000,C 90.000,E1 83.913} C_DIS
LIN {X -0.146,Y -400.738,Z 424.454,A 0.000,B 0.000,C 90.000,E1 81.724} C_DIS
LIN {X -0.064,Y -390.120,Z 424.443,A 0.000,B 0.000,C 90.000,E1 79.746} C_DIS
LIN {X -0.101,Y -378.141,Z 424.430,A 0.000,B 0.000,C 90.000,E1 77.465} C_DIS
LIN {X 0.092,Y -365.228,Z 424.416,A 0.000,B 0.000,C 90.000,E1 74.810} C_DIS
LIN {X 0.119,Y -349.061,Z 424.396,A 0.000,B 0.000,C 90.000,E1 71.221} C_DIS
LIN {X 0.150,Y -336.470,Z 424.379,A 0.000,B 0.000,C 90.000,E1 68.156} C_DIS
LIN {X 0.129,Y -326.671,Z 424.365,A 0.000,B 0.000,C 90.000,E1 65.665} C_DIS
LIN {X 0.135,Y -317.151,Z 424.351,A 0.000,B 0.000,C 90.000,E1 63.127} C_DIS
LIN {X 0.009,Y -305.583,Z 424.333,A 0.000,B 0.000,C 90.000,E1 59.921} C_DIS
LIN {X 0.016,Y -293.723,Z 424.313,A 0.000,B 0.000,C 90.000,E1 56.294} C_DIS
LIN {X 0.071,Y -283.937,Z 424.294,A 0.000,B 0.000,C 90.000,E1 52.924} C_DIS
LIN {X 0.063,Y -276.418,Z 424.279,A 0.000,B 0.000,C 90.000,E1 50.194} C_DIS
LIN {X -0.131,Y -270.648,Z 424.267,A 0.000,B 0.000,C 90.000,E1 48.162} C_DIS
LIN {X -0.073,Y -264.610,Z 424.256,A 0.000,B 0.000,C 90.000,E1 46.053} C_DIS
LIN {X -0.133,Y -258.458,Z 424.244,A 0.000,B 0.000,C 90.000,E1 43.947} C_DIS
LIN {X 0.060,Y -252.086,Z 424.232,A 0.000,B 0.000,C 90.000,E1 41.757} C_DIS
LIN {X -0.032,Y -243.518,Z 424.216,A 0.000,B 0.000,C 90.000,E1 38.874} C_DIS
LIN {X -0.070,Y -233.432,Z 424.195,A 0.000,B 0.000,C 90.000,E1 35.185} C_DIS
LIN {X 0.080,Y -226.176,Z 424.179,A 0.000,B 0.000,C 90.000,E1 32.133} C_DIS
LIN {X 0.065,Y -219.652,Z 424.162,A 0.000,B 0.000,C 90.000,E1 29.077} C_DIS
LIN {X 0.064,Y -213.793,Z 424.144,A 0.000,B 0.000,C 90.000,E1 25.976} C_DIS
LIN {X 0.034,Y -208.610,Z 424.127,A 0.000,B 0.000,C 90.000,E1 22.845} C_DIS
LIN {X -0.087,Y -202.978,Z 424.105,A 0.000,B 0.000,C 90.000,E1 18.906} C_DIS
LIN {X 0.116,Y -198.310,Z 424.083,A 0.000,B 0.000,C 90.000,E1 14.828} C_DIS
LIN {X 0.084,Y -193.966,Z 424.055,A 0.000,B 0.000,C 90.000,E1 9.962} C_DIS
LIN {X 0.061,Y -191.073,Z 424.028,A 0.000,B 0.000,C 90.000,E1 5.049} C_DIS
LIN {X -0.001,Y -189.626,Z 423.988,A 0.000,B 0.000,C 90.000,E1 357.879} C_DIS
LIN {X 0.017,Y -191.691,Z 423.947,A 0.000,B 0.000,C 90.000,E1 350.443} C_DIS
LIN {X 0.007,Y -194.813,Z 423.920,A 0.000,B 0.000,C 90.000,E1 345.519} C_DIS
LIN {X -0.046,Y -198.462,Z 423.897,A 0.000,B 0.000,C 90.000,E1 341.456} C_DIS
LIN {X -0.040,Y -203.135,Z 423.874,A 0.000,B 0.000,C 90.000,E1 337.411} C_DIS
LIN {X 0.058,Y -208.864,Z 423.852,A 0.000,B 0.000,C 90.000,E1 333.384} C_DIS
LIN {X -0.032,Y -215.419,Z 423.830,A 0.000,B 0.000,C 90.000,E1 329.459} C_DIS
LIN {X 0.037,Y -222.461,Z 423.809,A 0.000,B 0.000,C 90.000,E1 325.548} C_DIS
LIN {X -0.085,Y -230.195,Z 423.787,A 0.000,B 0.000,C 90.000,E1 321.743} C_DIS
LIN {X -0.033,Y -239.037,Z 423.766,A 0.000,B 0.000,C 90.000,E1 317.957} C_DIS
LIN {X 0.091,Y -248.004,Z 423.748,A 0.000,B 0.000,C 90.000,E1 314.595} C_DIS
LIN {X 0.140,Y -257.042,Z 423.732,A 0.000,B 0.000,C 90.000,E1 311.676} C_DIS
LIN {X 0.165,Y -268.360,Z 423.714,A 0.000,B 0.000,C 90.000,E1 308.463} C_DIS
LIN {X 0.013,Y -280.603,Z 423.696,A 0.000,B 0.000,C 90.000,E1 305.358} C_DIS
LIN {X 0.055,Y -290.707,Z 423.683,A 0.000,B 0.000,C 90.000,E1 302.959} C_DIS
LIN {X 0.176,Y -301.066,Z 423.670,A 0.000,B 0.000,C 90.000,E1 300.590} C_DIS
LIN {X 0.085,Y -317.179,Z 423.652,A 0.000,B 0.000,C 90.000,E1 297.334} C_DIS
LIN {X 0.087,Y -335.017,Z 423.634,A 0.000,B 0.000,C 90.000,E1 294.155} C_DIS
LIN {X -0.064,Y -355.601,Z 423.617,A 0.000,B 0.000,C 90.000,E1 291.099} C_DIS
LIN {X -0.068,Y -376.006,Z 423.602,A 0.000,B 0.000,C 90.000,E1 288.417} C_DIS
LIN {X -0.110,Y -387.849,Z 423.594,A 0.000,B 0.000,C 90.000,E1 286.985} C_DIS
LIN {X 0.123,Y -402.786,Z 423.585,A 0.000,B 0.000,C 90.000,E1 285.315} C_DIS
LIN {X -0.021,Y -421.037,Z 423.575,A 0.000,B 0.000,C 90.000,E1 283.536} C_DIS
LIN {X -0.109,Y -431.415,Z 423.570,A 0.000,B 0.000,C 90.000,E1 282.535} C_DIS
LIN {X 0.119,Y -441.368,Z 423.564,A 0.000,B 0.000,C 90.000,E1 281.478} C_DIS
LIN {X -0.072,Y -448.564,Z 423.559,A 0.000,B 0.000,C 90.000,E1 280.715} C_DIS
LIN {X 0.125,Y -455.198,Z 423.555,A 0.000,B 0.000,C 90.000,E1 279.905} C_DIS
LIN {X 0.223,Y -463.206,Z 423.549,A 0.000,B 0.000,C 90.000,E1 278.859} C_DIS
LIN {X -0.052,Y -470.267,Z 423.544,A 0.000,B 0.000,C 90.000,E1 277.871} C_DIS
LIN {X 0.155,Y -476.764,Z 423.538,A 0.000,B 0.000,C 90.000,E1 276.834} C_DIS
LIN {X 0.102,Y -481.138,Z 423.534,A 0.000,B 0.000,C 90.000,E1 276.087} C_DIS
LIN {X 0.134,Y -484.905,Z 423.530,A 0.000,B 0.000,C 90.000,E1 275.334} C_DIS
LIN {X -0.209,Y -487.004,Z 423.527,A 0.000,B 0.000,C 90.000,E1 274.878} C_DIS
LIN {X -0.011,Y -488.709,Z 423.524,A 0.000,B 0.000,C 90.000,E1 274.359} C_DIS
LIN {X 0.192,Y -490.062,Z 423.521,A 0.000,B 0.000,C 90.000,E1 273.841} C_DIS
LIN {X -0.117,Y -491.125,Z 423.519,A 0.000,B 0.000,C 90.000,E1 273.383} C_DIS
LIN {X 0.100,Y -491.851,Z 423.516,A 0.000,B 0.000,C 90.000,E1 272.865} C_DIS
LIN {X -0.193,Y -492.222,Z 423.513,A 0.000,B 0.000,C 90.000,E1 272.407} C_DIS
LIN {X 0.012,Y -492.145,Z 423.511,A 0.000,B 0.000,C 90.000,E1 271.892} C_DIS
LIN {X 0.234,Y -491.671,Z 423.508,A 0.000,B 0.000,C 90.000,E1 271.375} C_DIS
LIN {X -0.050,Y -490.733,Z 423.505,A 0.000,B 0.000,C 90.000,E1 270.917} C_DIS
LIN {X 0.155,Y -489.323,Z 423.502,A 0.000,B 0.000,C 90.000,E1 270.401} C_DIS
LIN {X -0.135,Y -487.335,Z 423.500,A 0.000,B 0.000,C 90.000,E1 269.943} C_DIS
LIN {X 0.056,Y -484.772,Z 423.497,A 0.000,B 0.000,C 90.000,E1 269.427} C_DIS
LIN {X 0.226,Y -481.558,Z 423.494,A 0.000,B 0.000,C 90.000,E1 268.912} C_DIS
LIN {X -0.102,Y -477.408,Z 423.491,A 0.000,B 0.000,C 90.000,E1 268.453} C_DIS
LIN {X 0.200,Y -474.968,Z 423.490,A 0.000,B 0.000,C 90.000,E1 268.167} C_DIS
LIN {X 0.043,Y -469.422,Z 423.487,A 0.000,B 0.000,C 90.000,E1 267.707} C_DIS
LIN {X -0.162,Y -463.132,Z 423.485,A 0.000,B 0.000,C 90.000,E1 267.306} C_DIS
LIN {X 0.170,Y -456.244,Z 423.483,A 0.000,B 0.000,C 90.000,E1 266.906} C_DIS
LIN {X 0.153,Y -449.184,Z 423.481,A 0.000,B 0.000,C 90.000,E1 266.617} C_DIS
LIN {X 0.112,Y -441.886,Z 423.480,A 0.000,B 0.000,C 90.000,E1 266.388} C_DIS
LIN {X -0.003,Y -434.254,Z 423.479,A 0.000,B 0.000,C 90.000,E1 266.216} C_DIS
LIN {X -0.208,Y -425.850,Z 423.478,A 0.000,B 0.000,C 90.000,E1 266.102} C_DIS
LIN {X -0.115,Y -414.814,Z 423.478,A 0.000,B 0.000,C 90.000,E1 265.988} C_DIS
LIN {X 0.145,Y -410.960,Z 423.478,A 0.000,B 0.000,C 90.000,E1 265.931} C_DIS
LIN {X 0.043,Y -180.918,Z 423.477,A 0.000,B 0.000,C 90.000,E1 265.927} C_DIS
LIN {X 0.073,Y -180.841,Z 423.472,A 0.000,B 0.000,C 90.000,E1 264.894} C_DIS
LIN {X -0.030,Y -178.883,Z 423.443,A 0.000,B 0.000,C 90.000,E1 259.690} C_DIS
LIN {X 0.046,Y -175.926,Z 423.414,A 0.000,B 0.000,C 90.000,E1 254.574} C_DIS
LIN {X -0.009,Y -175.365,Z 423.410,A 0.000,B 0.000,C 90.000,E1 253.740} C_DIS
LIN {X 0.050,Y -172.143,Z 423.386,A 0.000,B 0.000,C 90.000,E1 249.444} C_DIS
LIN {X 0.027,Y -171.607,Z 423.381,A 0.000,B 0.000,C 90.000,E1 248.592} C_DIS
LIN {X 0.015,Y -167.830,Z 423.357,A 0.000,B 0.000,C 90.000,E1 244.280} C_DIS
LIN {X 0.032,Y -166.556,Z 423.348,A 0.000,B 0.000,C 90.000,E1 242.538} C_DIS
LIN {X -0.057,Y -162.551,Z 423.323,A 0.000,B 0.000,C 90.000,E1 238.201} C_DIS
LIN {X 0.002,Y -161.229,Z 423.313,A 0.000,B 0.000,C 90.000,E1 236.421} C_DIS
LIN {X 0.038,Y -157.234,Z 423.289,A 0.000,B 0.000,C 90.000,E1 231.984} C_DIS
LIN {X 0.060,Y -155.958,Z 423.279,A 0.000,B 0.000,C 90.000,E1 230.194} C_DIS
LIN {X 0.019,Y -152.212,Z 423.254,A 0.000,B 0.000,C 90.000,E1 225.729} C_DIS
LIN {X 0.040,Y -150.457,Z 423.239,A 0.000,B 0.000,C 90.000,E1 223.014} C_DIS
LIN {X 0.066,Y -147.182,Z 423.214,A 0.000,B 0.000,C 90.000,E1 218.463} C_DIS
LIN {X 0.032,Y -145.200,Z 423.194,A 0.000,B 0.000,C 90.000,E1 214.818} C_DIS
LIN {X -0.058,Y -142.337,Z 423.163,A 0.000,B 0.000,C 90.000,E1 209.333} C_DIS
LIN {X -0.005,Y -141.726,Z 423.153,A 0.000,B 0.000,C 90.000,E1 207.462} C_DIS
LIN {X -0.022,Y -139.480,Z 423.116,A 0.000,B 0.000,C 90.000,E1 200.972} C_DIS
LIN {X -0.033,Y -138.978,Z 423.101,A 0.000,B 0.000,C 90.000,E1 198.181} C_DIS
LIN {X -0.048,Y -138.332,Z 423.054,A 0.000,B 0.000,C 90.000,E1 189.782} C_DIS
LIN {X -0.048,Y -139.430,Z 423.008,A 0.000,B 0.000,C 90.000,E1 181.375} C_DIS
LIN {X 0.005,Y -141.357,Z 422.971,A 0.000,B 0.000,C 90.000,E1 174.837} C_DIS
LIN {X -0.018,Y -142.711,Z 422.956,A 0.000,B 0.000,C 90.000,E1 172.064} C_DIS
LIN {X -0.059,Y -145.086,Z 422.930,A 0.000,B 0.000,C 90.000,E1 167.465} C_DIS
LIN {X -0.064,Y -147.711,Z 422.910,A 0.000,B 0.000,C 90.000,E1 163.795} C_DIS
LIN {X 0.019,Y -150.366,Z 422.890,A 0.000,B 0.000,C 90.000,E1 160.115} C_DIS
LIN {X 0.038,Y -153.793,Z 422.869,A 0.000,B 0.000,C 90.000,E1 156.485} C_DIS
LIN {X -0.042,Y -157.204,Z 422.849,A 0.000,B 0.000,C 90.000,E1 152.922} C_DIS
LIN {X 0.039,Y -161.368,Z 422.830,A 0.000,B 0.000,C 90.000,E1 149.331} C_DIS
LIN {X 0.050,Y -165.570,Z 422.810,A 0.000,B 0.000,C 90.000,E1 145.801} C_DIS
LIN {X -0.067,Y -170.489,Z 422.791,A 0.000,B 0.000,C 90.000,E1 142.351} C_DIS
LIN {X 0.083,Y -175.369,Z 422.772,A 0.000,B 0.000,C 90.000,E1 138.852} C_DIS
LIN {X -0.055,Y -180.994,Z 422.753,A 0.000,B 0.000,C 90.000,E1 135.486} C_DIS
LIN {X 0.070,Y -186.420,Z 422.734,A 0.000,B 0.000,C 90.000,E1 132.081} C_DIS
LIN {X 0.018,Y -191.047,Z 422.720,A 0.000,B 0.000,C 90.000,E1 129.600} C_DIS
LIN {X 0.069,Y -196.435,Z 422.703,A 0.000,B 0.000,C 90.000,E1 126.503} C_DIS
LIN {X 0.062,Y -294.416,Z 422.703,A 0.000,B 0.000,C 90.000,E1 126.503} C_DIS
LIN {X 0.095,Y -300.642,Z 422.702,A 0.000,B 0.000,C 90.000,E1 126.297} C_DIS
LIN {X 0.112,Y -303.242,Z 422.701,A 0.000,B 0.000,C 90.000,E1 126.091} C_DIS
LIN {X 0.025,Y -307.055,Z 422.698,A 0.000,B 0.000,C 90.000,E1 125.644} C_DIS
LIN {X 0.063,Y -308.925,Z 422.696,A 0.000,B 0.000,C 90.000,E1 125.311} C_DIS
LIN {X -0.153,Y -310.389,Z 422.694,A 0.000,B 0.000,C 90.000,E1 125.025} C_DIS
LIN {X -0.048,Y -314.645,Z 422.687,A 0.000,B 0.000,C 90.000,E1 123.706} C_DIS
LIN {X 0.077,Y -324.782,Z 422.671,A 0.000,B 0.000,C 90.000,E1 120.797} C_DIS
LIN {X 0.001,Y -336.262,Z 422.655,A 0.000,B 0.000,C 90.000,E1 117.975} C_DIS
LIN {X -0.063,Y -349.182,Z 422.640,A 0.000,B 0.000,C 90.000,E1 115.207} C_DIS
LIN {X 0.054,Y -361.974,Z 422.627,A 0.000,B 0.000,C 90.000,E1 112.770} C_DIS
LIN {X -0.117,Y -376.093,Z 422.613,A 0.000,B 0.000,C 90.000,E1 110.429} C_DIS
LIN {X -0.079,Y -391.641,Z 422.601,A 0.000,B 0.000,C 90.000,E1 108.109} C_DIS
LIN {X -0.016,Y -408.733,Z 422.588,A 0.000,B 0.000,C 90.000,E1 105.843} C_DIS
LIN {X -0.029,Y -427.496,Z 422.576,A 0.000,B 0.000,C 90.000,E1 103.647} C_DIS
LIN {X 0.206,Y -447.521,Z 422.564,A 0.000,B 0.000,C 90.000,E1 101.535} C_DIS
LIN {X -0.144,Y -468.118,Z 422.554,A 0.000,B 0.000,C 90.000,E1 99.670} C_DIS
LIN {X 0.033,Y -486.455,Z 422.545,A 0.000,B 0.000,C 90.000,E1 98.106} C_DIS
LIN {X -0.237,Y -490.024,Z 422.543,A 0.000,B 0.000,C 90.000,E1 97.701} C_DIS
LIN {X 0.139,Y -491.370,Z 422.541,A 0.000,B 0.000,C 90.000,E1 97.409} C_DIS
LIN {X -0.035,Y -492.363,Z 422.540,A 0.000,B 0.000,C 90.000,E1 97.182} C_DIS
LIN {X 0.198,Y -493.475,Z 422.537,A 0.000,B 0.000,C 90.000,E1 96.663} C_DIS
LIN {X -0.053,Y -493.575,Z 422.534,A 0.000,B 0.000,C 90.000,E1 96.201} C_DIS
LIN {X 0.192,Y -492.674,Z 422.532,A 0.000,B 0.000,C 90.000,E1 95.682} C_DIS
LIN {X -0.054,Y -490.613,Z 422.529,A 0.000,B 0.000,C 90.000,E1 95.220} C_DIS
LIN {X -0.202,Y -489.012,Z 422.528,A 0.000,B 0.000,C 90.000,E1 94.992} C_DIS
LIN {X 0.061,Y -479.304,Z 422.521,A 0.000,B 0.000,C 90.000,E1 93.726} C_DIS
LIN {X 0.108,Y -455.878,Z 422.504,A 0.000,B 0.000,C 90.000,E1 90.688} C_DIS
LIN {X 0.102,Y -436.703,Z 422.488,A 0.000,B 0.000,C 90.000,E1 87.822} C_DIS
LIN {X 0.081,Y -417.261,Z 422.470,A 0.000,B 0.000,C 90.000,E1 84.609} C_DIS
LIN {X 0.086,Y -404.941,Z 422.458,A 0.000,B 0.000,C 90.000,E1 82.413} C_DIS
LIN {X -0.127,Y -392.751,Z 422.445,A 0.000,B 0.000,C 90.000,E1 80.208} C_DIS
LIN {X -0.173,Y -380.736,Z 422.433,A 0.000,B 0.000,C 90.000,E1 77.937} C_DIS
LIN {X 0.078,Y -366.299,Z 422.417,A 0.000,B 0.000,C 90.000,E1 74.991} C_DIS
LIN {X 0.142,Y -350.023,Z 422.397,A 0.000,B 0.000,C 90.000,E1 71.402} C_DIS
LIN {X 0.076,Y -337.351,Z 422.380,A 0.000,B 0.000,C 90.000,E1 68.358} C_DIS
LIN {X 0.101,Y -328.735,Z 422.368,A 0.000,B 0.000,C 90.000,E1 66.177} C_DIS
LIN {X 0.090,Y -317.921,Z 422.352,A 0.000,B 0.000,C 90.000,E1 63.332} C_DIS
LIN {X -0.019,Y -306.308,Z 422.334,A 0.000,B 0.000,C 90.000,E1 60.127} C_DIS
LIN {X 0.011,Y -294.363,Z 422.314,A 0.000,B 0.000,C 90.000,E1 56.501} C_DIS
LIN {X 0.088,Y -284.540,Z 422.295,A 0.000,B 0.000,C 90.000,E1 53.130} C_DIS
LIN {X -0.080,Y -277.016,Z 422.280,A 0.000,B 0.000,C 90.000,E1 50.436} C_DIS
LIN {X 0.119,Y -271.282,Z 422.269,A 0.000,B 0.000,C 90.000,E1 48.324} C_DIS
LIN {X -0.008,Y -265.276,Z 422.257,A 0.000,B 0.000,C 90.000,E1 46.257} C_DIS
LIN {X 0.128,Y -259.157,Z 422.245,A 0.000,B 0.000,C 90.000,E1 44.109} C_DIS
LIN {X -0.027,Y -252.823,Z 422.233,A 0.000,B 0.000,C 90.000,E1 42.000} C_DIS
LIN {X -0.093,Y -244.280,Z 422.217,A 0.000,B 0.000,C 90.000,E1 39.116} C_DIS
LIN {X 0.037,Y -234.139,Z 422.197,A 0.000,B 0.000,C 90.000,E1 35.391} C_DIS
LIN {X -0.112,Y -226.806,Z 422.180,A 0.000,B 0.000,C 90.000,E1 32.418} C_DIS
LIN {X 0.009,Y -220.211,Z 422.163,A 0.000,B 0.000,C 90.000,E1 29.333} C_DIS
LIN {X 0.023,Y -214.288,Z 422.146,A 0.000,B 0.000,C 90.000,E1 26.232} C_DIS
LIN {X 0.087,Y -209.026,Z 422.128,A 0.000,B 0.000,C 90.000,E1 23.078} C_DIS
LIN {X -0.030,Y -203.312,Z 422.106,A 0.000,B 0.000,C 90.000,E1 19.141} C_DIS
LIN {X -0.064,Y -198.561,Z 422.084,A 0.000,B 0.000,C 90.000,E1 15.134} C_DIS
LIN {X -0.035,Y -194.123,Z 422.057,A 0.000,B 0.000,C 90.000,E1 10.254} C_DIS
LIN {X -0.031,Y -191.101,Z 422.030,A 0.000,B 0.000,C 90.000,E1 5.334} C_DIS
LIN {X -0.002,Y -189.536,Z 421.988,A 0.000,B 0.000,C 90.000,E1 357.879} C_DIS
LIN {X 0.011,Y -191.582,Z 421.947,A 0.000,B 0.000,C 90.000,E1 350.443} C_DIS
LIN {X -0.004,Y -194.693,Z 421.920,A 0.000,B 0.000,C 90.000,E1 345.519} C_DIS
LIN {X -0.062,Y -198.331,Z 421.897,A 0.000,B 0.000,C 90.000,E1 341.456} C_DIS
LIN {X -0.060,Y -202.992,Z 421.874,A 0.000,B 0.000,C 90.000,E1 337.411} C_DIS
LIN {X -0.053,Y -207.488,Z 421.857,A 0.000,B 0.000,C 90.000,E1 334.204} C_DIS
LIN {X 0.085,Y -213.919,Z 421.835,A 0.000,B 0.000,C 90.000,E1 330.205} C_DIS
LIN {X 0.108,Y -220.870,Z 421.813,A 0.000,B 0.000,C 90.000,E1 326.294} C_DIS
LIN {X -0.012,Y -228.425,Z 421.792,A 0.000,B 0.000,C 90.000,E1 322.477} C_DIS
LIN {X -0.011,Y -237.050,Z 421.770,A 0.000,B 0.000,C 90.000,E1 318.690} C_DIS
LIN {X 0.062,Y -245.818,Z 421.752,A 0.000,B 0.000,C 90.000,E1 315.324} C_DIS
LIN {X -0.132,Y -254.582,Z 421.736,A 0.000,B 0.000,C 90.000,E1 312.447} C_DIS
LIN {X -0.021,Y -265.653,Z 421.718,A 0.000,B 0.000,C 90.000,E1 309.197} C_DIS
LIN {X 0.036,Y -276.403,Z 421.702,A 0.000,B 0.000,C 90.000,E1 306.377} C_DIS
LIN {X 0.011,Y -289.184,Z 421.685,A 0.000,B 0.000,C 90.000,E1 303.293} C_DIS
LIN {X -0.020,Y -304.106,Z 421.666,A 0.000,B 0.000,C 90.000,E1 299.951} C_DIS
LIN {X -0.012,Y -320.595,Z 421.648,A 0.000,B 0.000,C 90.000,E1 296.693} C_DIS
LIN {X 0.001,Y -335.054,Z 421.634,A 0.000,B 0.000,C 90.000,E1 294.155} C_DIS
LIN {X -0.188,Y -353.532,Z 421.619,A 0.000,B 0.000,C 90.000,E1 291.408} C_DIS
LIN {X 0.133,Y -371.498,Z 421.605,A 0.000,B 0.000,C 90.000,E1 288.960} C_DIS
LIN {X 0.227,Y -388.088,Z 421.594,A 0.000,B 0.000,C 90.000,E1 286.913} C_DIS
LIN {X -0.013,Y -403.063,Z 421.585,A 0.000,B 0.000,C 90.000,E1 285.315} C_DIS
LIN {X -0.237,Y -421.443,Z 421.575,A 0.000,B 0.000,C 90.000,E1 283.536} C_DIS
LIN {X 0.118,Y -431.740,Z 421.569,A 0.000,B 0.000,C 90.000,E1 282.479} C_DIS
LIN {X -0.068,Y -441.686,Z 421.564,A 0.000,B 0.000,C 90.000,E1 281.478} C_DIS
LIN {X 0.165,Y -448.842,Z 421.559,A 0.000,B 0.000,C 90.000,E1 280.658} C_DIS
LIN {X -0.077,Y -455.444,Z 421.555,A 0.000,B 0.000,C 90.000,E1 279.905} C_DIS
LIN {X 0.199,Y -461.487,Z 421.551,A 0.000,B 0.000,C 90.000,E1 279.095} C_DIS
LIN {X 0.070,Y -466.998,Z 421.546,A 0.000,B 0.000,C 90.000,E1 278.341} C_DIS
LIN {X -0.164,Y -473.757,Z 421.541,A 0.000,B 0.000,C 90.000,E1 277.352} C_DIS
LIN {X -0.248,Y -478.403,Z 421.537,A 0.000,B 0.000,C 90.000,E1 276.606} C_DIS
LIN {X 0.239,Y -482.582,Z 421.532,A 0.000,B 0.000,C 90.000,E1 275.796} C_DIS
LIN {X -0.072,Y -485.012,Z 421.530,A 0.000,B 0.000,C 90.000,E1 275.334} C_DIS
LIN {X 0.070,Y -487.026,Z 421.527,A 0.000,B 0.000,C 90.000,E1 274.821} C_DIS
LIN {X -0.223,Y -488.756,Z 421.524,A 0.000,B 0.000,C 90.000,E1 274.359} C_DIS
LIN {X -0.021,Y -490.118,Z 421.521,A 0.000,B 0.000,C 90.000,E1 273.841} C_DIS
LIN {X 0.160,Y -491.134,Z 421.519,A 0.000,B 0.000,C 90.000,E1 273.326} C_DIS
LIN {X -0.113,Y -491.844,Z 421.516,A 0.000,B 0.000,C 90.000,E1 272.865} C_DIS
LIN {X 0.085,Y -492.213,Z 421.513,A 0.000,B 0.000,C 90.000,E1 272.350} C_DIS
LIN {X -0.201,Y -492.156,Z 421.510,A 0.000,B 0.000,C 90.000,E1 271.892} C_DIS
LIN {X 0.021,Y -491.641,Z 421.508,A 0.000,B 0.000,C 90.000,E1 271.375} C_DIS
LIN {X 0.228,Y -490.724,Z 421.505,A 0.000,B 0.000,C 90.000,E1 270.859} C_DIS
LIN {X -0.058,Y -489.285,Z 421.502,A 0.000,B 0.000,C 90.000,E1 270.401} C_DIS
LIN {X 0.142,Y -487.287,Z 421.499,A 0.000,B 0.000,C 90.000,E1 269.885} C_DIS
LIN {X -0.154,Y -484.709,Z 421.497,A 0.000,B 0.000,C 90.000,E1 269.427} C_DIS
LIN {X 0.017,Y -481.435,Z 421.494,A 0.000,B 0.000,C 90.000,E1 268.912} C_DIS
LIN {X -0.147,Y -479.475,Z 421.493,A 0.000,B 0.000,C 90.000,E1 268.682} C_DIS
LIN {X 0.008,Y -474.802,Z 421.490,A 0.000,B 0.000,C 90.000,E1 268.165} C_DIS
LIN {X -0.159,Y -469.149,Z 421.487,A 0.000,B 0.000,C 90.000,E1 267.707} C_DIS
LIN {X -0.156,Y -465.982,Z 421.486,A 0.000,B 0.000,C 90.000,E1 267.478} C_DIS
LIN {X -0.136,Y -459.122,Z 421.484,A 0.000,B 0.000,C 90.000,E1 267.078} C_DIS
LIN {X 0.052,Y -451.850,Z 421.482,A 0.000,B 0.000,C 90.000,E1 266.731} C_DIS
LIN {X -0.150,Y -444.685,Z 421.480,A 0.000,B 0.000,C 90.000,E1 266.502} C_DIS
LIN {X 0.036,Y -437.061,Z 421.479,A 0.000,B 0.000,C 90.000,E1 266.274} C_DIS
LIN {X 0.153,Y -429.274,Z 421.478,A 0.000,B 0.000,C 90.000,E1 266.102} C_DIS
LIN {X 0.108,Y -419.318,Z 421.478,A 0.000,B 0.000,C 90.000,E1 265.988} C_DIS
LIN {X 0.121,Y -407.270,Z 421.477,A 0.000,B 0.000,C 90.000,E1 265.927} C_DIS
LIN {X 0.022,Y -180.917,Z 421.477,A 0.000,B 0.000,C 90.000,E1 265.927} C_DIS
LIN {X 0.054,Y -180.839,Z 421.472,A 0.000,B 0.000,C 90.000,E1 264.894} C_DIS
LIN {X -0.049,Y -178.880,Z 421.443,A 0.000,B 0.000,C 90.000,E1 259.690} C_DIS
LIN {X 0.027,Y -175.923,Z 421.414,A 0.000,B 0.000,C 90.000,E1 254.574} C_DIS
LIN {X -0.028,Y -175.359,Z 421.410,A 0.000,B 0.000,C 90.000,E1 253.740} C_DIS
LIN {X 0.031,Y -172.139,Z 421.386,A 0.000,B 0.000,C 90.000,E1 249.444} C_DIS
LIN {X 0.009,Y -171.602,Z 421.381,A 0.000,B 0.000,C 90.000,E1 248.592} C_DIS
LIN {X -0.003,Y -167.825,Z 421.357,A 0.000,B 0.000,C 90.000,E1 244.280} C_DIS
LIN {X 0.014,Y -166.550,Z 421.347,A 0.000,B 0.000,C 90.000,E1 242.538} C_DIS
LIN {X -0.074,Y -162.546,Z 421.323,A 0.000,B 0.000,C 90.000,E1 238.201} C_DIS
LIN {X -0.015,Y -161.223,Z 421.313,A 0.000,B 0.000,C 90.000,E1 236.421} C_DIS
LIN {X 0.021,Y -157.230,Z 421.289,A 0.000,B 0.000,C 90.000,E1 231.984} C_DIS
LIN {X 0.043,Y -155.954,Z 421.279,A 0.000,B 0.000,C 90.000,E1 230.194} C_DIS
LIN {X 0.002,Y -152.208,Z 421.254,A 0.000,B 0.000,C 90.000,E1 225.729} C_DIS
LIN {X 0.023,Y -150.452,Z 421.239,A 0.000,B 0.000,C 90.000,E1 223.014} C_DIS
LIN {X 0.050,Y -147.178,Z 421.214,A 0.000,B 0.000,C 90.000,E1 218.463} C_DIS
LIN {X 0.017,Y -145.195,Z 421.193,A 0.000,B 0.000,C 90.000,E1 214.818} C_DIS
LIN {X 0.050,Y -142.335,Z 421.163,A 0.000,B 0.000,C 90.000,E1 209.283} C_DIS
LIN {X -0.020,Y -141.724,Z 421.153,A 0.000,B 0.000,C 90.000,E1 207.462} C_DIS
LIN {X -0.038,Y -139.479,Z 421.116,A 0.000,B 0.000,C 90.000,E1 200.972} C_DIS
LIN {X -0.048,Y -138.976,Z 421.101,A 0.000,B 0.000,C 90.000,E1 198.181} C_DIS
LIN {X 0.073,Y -138.332,Z 421.054,A 0.000,B 0.000,C 90.000,E1 189.726} C_DIS
LIN {X -0.063,Y -139.432,Z 421.008,A 0.000,B 0.000,C 90.000,E1 181.375} C_DIS
LIN {X 0.016,Y -140.958,Z 420.976,A 0.000,B 0.000,C 90.000,E1 175.755} C_DIS
LIN {X -0.033,Y -142.713,Z 420.956,A 0.000,B 0.000,C 90.000,E1 172.064} C_DIS
LIN {X 0.066,Y -145.090,Z 420.930,A 0.000,B 0.000,C 90.000,E1 167.409} C_DIS
LIN {X 0.061,Y -147.714,Z 420.910,A 0.000,B 0.000,C 90.000,E1 163.740} C_DIS
LIN {X 0.003,Y -150.372,Z 420.890,A 0.000,B 0.000,C 90.000,E1 160.115} C_DIS
LIN {X 0.021,Y -153.799,Z 420.869,A 0.000,B 0.000,C 90.000,E1 156.485} C_DIS
LIN {X 0.081,Y -157.211,Z 420.849,A 0.000,B 0.000,C 90.000,E1 152.871} C_DIS
LIN {X 0.022,Y -161.376,Z 420.830,A 0.000,B 0.000,C 90.000,E1 149.331} C_DIS
LIN {X 0.033,Y -165.578,Z 420.810,A 0.000,B 0.000,C 90.000,E1 145.801} C_DIS
LIN {X 0.020,Y -170.497,Z 420.791,A 0.000,B 0.000,C 90.000,E1 142.316} C_DIS
LIN {X 0.064,Y -175.378,Z 420.772,A 0.000,B 0.000,C 90.000,E1 138.852} C_DIS
LIN {X -0.073,Y -181.002,Z 420.753,A 0.000,B 0.000,C 90.000,E1 135.486} C_DIS
LIN {X 0.051,Y -186.430,Z 420.734,A 0.000,B 0.000,C 90.000,E1 132.081} C_DIS
LIN {X 0.121,Y -191.056,Z 420.720,A 0.000,B 0.000,C 90.000,E1 129.564} C_DIS
LIN {X 0.033,Y -196.542,Z 420.703,A 0.000,B 0.000,C 90.000,E1 126.457} C_DIS
LIN {X 0.015,Y -295.373,Z 420.703,A 0.000,B 0.000,C 90.000,E1 126.457} C_DIS
LIN {X 0.066,Y -300.020,Z 420.702,A 0.000,B 0.000,C 90.000,E1 126.297} C_DIS
LIN {X -0.009,Y -303.073,Z 420.701,A 0.000,B 0.000,C 90.000,E1 126.091} C_DIS
LIN {X 0.066,Y -306.800,Z 420.698,A 0.000,B 0.000,C 90.000,E1 125.644} C_DIS
LIN {X 0.158,Y -308.705,Z 420.696,A 0.000,B 0.000,C 90.000,E1 125.311} C_DIS
LIN {X 0.000,Y -310.202,Z 420.695,A 0.000,B 0.000,C 90.000,E1 125.025} C_DIS
LIN {X -0.173,Y -312.456,Z 420.691,A 0.000,B 0.000,C 90.000,E1 124.405} C_DIS
LIN {X 0.057,Y -322.296,Z 420.675,A 0.000,B 0.000,C 90.000,E1 121.465} C_DIS
LIN {X 0.069,Y -333.455,Z 420.659,A 0.000,B 0.000,C 90.000,E1 118.615} C_DIS
LIN {X -0.075,Y -346.031,Z 420.644,A 0.000,B 0.000,C 90.000,E1 115.848} C_DIS
LIN {X 0.107,Y -358.493,Z 420.630,A 0.000,B 0.000,C 90.000,E1 113.387} C_DIS
LIN {X -0.150,Y -372.256,Z 420.617,A 0.000,B 0.000,C 90.000,E1 111.046} C_DIS
LIN {X -0.203,Y -387.421,Z 420.604,A 0.000,B 0.000,C 90.000,E1 108.725} C_DIS
LIN {X -0.128,Y -404.099,Z 420.591,A 0.000,B 0.000,C 90.000,E1 106.441} C_DIS
LIN {X 0.152,Y -422.413,Z 420.579,A 0.000,B 0.000,C 90.000,E1 104.189} C_DIS
LIN {X 0.180,Y -442.218,Z 420.567,A 0.000,B 0.000,C 90.000,E1 102.063} C_DIS
LIN {X -0.062,Y -462.677,Z 420.556,A 0.000,B 0.000,C 90.000,E1 100.141} C_DIS
LIN {X 0.180,Y -486.262,Z 420.545,A 0.000,B 0.000,C 90.000,E1 98.106} C_DIS
LIN {X -0.037,Y -489.955,Z 420.543,A 0.000,B 0.000,C 90.000,E1 97.701} C_DIS
LIN {X -0.148,Y -491.364,Z 420.541,A 0.000,B 0.000,C 90.000,E1 97.466} C_DIS
LIN {X 0.165,Y -492.411,Z 420.540,A 0.000,B 0.000,C 90.000,E1 97.182} C_DIS
LIN {X -0.091,Y -493.610,Z 420.537,A 0.000,B 0.000,C 90.000,E1 96.720} C_DIS
LIN {X 0.148,Y -493.786,Z 420.535,A 0.000,B 0.000,C 90.000,E1 96.201} C_DIS
LIN {X -0.097,Y -492.967,Z 420.532,A 0.000,B 0.000,C 90.000,E1 95.739} C_DIS
LIN {X 0.147,Y -491.012,Z 420.529,A 0.000,B 0.000,C 90.000,E1 95.220} C_DIS
LIN {X 0.001,Y -489.485,Z 420.528,A 0.000,B 0.000,C 90.000,E1 94.992} C_DIS
LIN {X -0.052,Y -481.804,Z 420.522,A 0.000,B 0.000,C 90.000,E1 94.012} C_DIS
LIN {X -0.036,Y -465.883,Z 420.511,A 0.000,B 0.000,C 90.000,E1 92.007} C_DIS
LIN {X 0.090,Y -450.916,Z 420.500,A 0.000,B 0.000,C 90.000,E1 89.943} C_DIS
LIN {X -0.063,Y -432.129,Z 420.484,A 0.000,B 0.000,C 90.000,E1 87.078} C_DIS
LIN {X -0.092,Y -411.479,Z 420.464,A 0.000,B 0.000,C 90.000,E1 83.571} C_DIS
LIN {X -0.216,Y -399.197,Z 420.452,A 0.000,B 0.000,C 90.000,E1 81.376} C_DIS
LIN {X -0.112,Y -387.109,Z 420.439,A 0.000,B 0.000,C 90.000,E1 79.106} C_DIS
LIN {X -0.117,Y -372.369,Z 420.423,A 0.000,B 0.000,C 90.000,E1 76.228} C_DIS
LIN {X 0.017,Y -359.697,Z 420.409,A 0.000,B 0.000,C 90.000,E1 73.559} C_DIS
LIN {X 0.026,Y -346.447,Z 420.392,A 0.000,B 0.000,C 90.000,E1 70.550} C_DIS
LIN {X -0.011,Y -335.163,Z 420.377,A 0.000,B 0.000,C 90.000,E1 67.794} C_DIS
LIN {X 0.029,Y -324.121,Z 420.361,A 0.000,B 0.000,C 90.000,E1 64.973} C_DIS
LIN {X 0.034,Y -313.381,Z 420.345,A 0.000,B 0.000,C 90.000,E1 62.103} C_DIS
LIN {X -0.087,Y -303.110,Z 420.329,A 0.000,B 0.000,C 90.000,E1 59.203} C_DIS
LIN {X 0.001,Y -292.477,Z 420.310,A 0.000,B 0.000,C 90.000,E1 55.881} C_DIS
LIN {X 0.014,Y -282.785,Z 420.292,A 0.000,B 0.000,C 90.000,E1 52.512} C_DIS
LIN {X -0.028,Y -275.274,Z 420.277,A 0.000,B 0.000,C 90.000,E1 49.784} C_DIS
LIN {X -0.069,Y -269.468,Z 420.265,A 0.000,B 0.000,C 90.000,E1 47.715} C_DIS
LIN {X 0.145,Y -263.422,Z 420.253,A 0.000,B 0.000,C 90.000,E1 45.567} C_DIS
LIN {X 0.058,Y -257.277,Z 420.242,A 0.000,B 0.000,C 90.000,E1 43.461} C_DIS
LIN {X 0.054,Y -250.888,Z 420.230,A 0.000,B 0.000,C 90.000,E1 41.310} C_DIS
LIN {X 0.124,Y -242.432,Z 420.213,A 0.000,B 0.000,C 90.000,E1 38.382} C_DIS
LIN {X 0.057,Y -234.388,Z 420.197,A 0.000,B 0.000,C 90.000,E1 35.438} C_DIS
LIN {X 0.051,Y -225.308,Z 420.176,A 0.000,B 0.000,C 90.000,E1 31.671} C_DIS
LIN {X 0.017,Y -218.851,Z 420.159,A 0.000,B 0.000,C 90.000,E1 28.615} C_DIS
LIN {X -0.097,Y -213.064,Z 420.142,A 0.000,B 0.000,C 90.000,E1 25.540} C_DIS
LIN {X -0.061,Y -207.930,Z 420.124,A 0.000,B 0.000,C 90.000,E1 22.386} C_DIS
LIN {X -0.090,Y -202.355,Z 420.102,A 0.000,B 0.000,C 90.000,E1 18.417} C_DIS
LIN {X 0.036,Y -197.777,Z 420.080,A 0.000,B 0.000,C 90.000,E1 14.356} C_DIS
LIN {X -0.050,Y -193.505,Z 420.053,A 0.000,B 0.000,C 90.000,E1 9.500} C_DIS
LIN {X 0.037,Y -190.353,Z 420.021,A 0.000,B 0.000,C 90.000,E1 3.726} C_DIS
LIN {X -0.049,Y -189.722,Z 419.974,A 0.000,B 0.000,C 90.000,E1 355.412} C_DIS
LIN {X -0.052,Y -192.348,Z 419.938,A 0.000,B 0.000,C 90.000,E1 348.814} C_DIS
LIN {X 0.045,Y -195.875,Z 419.910,A 0.000,B 0.000,C 90.000,E1 343.866} C_DIS
LIN {X -0.051,Y -199.936,Z 419.888,A 0.000,B 0.000,C 90.000,E1 339.826} C_DIS
LIN {X -0.040,Y -205.004,Z 419.865,A 0.000,B 0.000,C 90.000,E1 335.793} C_DIS
LIN {X 0.110,Y -211.149,Z 419.843,A 0.000,B 0.000,C 90.000,E1 331.769} C_DIS
LIN {X 0.008,Y -217.889,Z 419.822,A 0.000,B 0.000,C 90.000,E1 327.867} C_DIS
LIN {X 0.027,Y -225.171,Z 419.800,A 0.000,B 0.000,C 90.000,E1 323.989} C_DIS
LIN {X 0.052,Y -231.625,Z 419.783,A 0.000,B 0.000,C 90.000,E1 320.928} C_DIS
LIN {X 0.033,Y -238.770,Z 419.766,A 0.000,B 0.000,C 90.000,E1 317.919} C_DIS
LIN {X -0.013,Y -247.790,Z 419.748,A 0.000,B 0.000,C 90.000,E1 314.595} C_DIS
LIN {X 0.026,Y -256.873,Z 419.732,A 0.000,B 0.000,C 90.000,E1 311.676} C_DIS
LIN {X 0.041,Y -268.228,Z 419.714,A 0.000,B 0.000,C 90.000,E1 308.463} C_DIS
LIN {X 0.109,Y -280.494,Z 419.696,A 0.000,B 0.000,C 90.000,E1 305.311} C_DIS
LIN {X -0.058,Y -289.130,Z 419.685,A 0.000,B 0.000,C 90.000,E1 303.293} C_DIS
LIN {X 0.058,Y -304.031,Z 419.666,A 0.000,B 0.000,C 90.000,E1 299.922} C_DIS
LIN {X 0.051,Y -320.556,Z 419.648,A 0.000,B 0.000,C 90.000,E1 296.668} C_DIS
LIN {X 0.052,Y -335.078,Z 419.634,A 0.000,B 0.000,C 90.000,E1 294.131} C_DIS
LIN {X 0.089,Y -355.793,Z 419.617,A 0.000,B 0.000,C 90.000,E1 291.046} C_DIS
LIN {X 0.106,Y -376.274,Z 419.602,A 0.000,B 0.000,C 90.000,E1 288.362} C_DIS
LIN {X 0.226,Y -388.146,Z 419.594,A 0.000,B 0.000,C 90.000,E1 286.913} C_DIS
LIN {X 0.016,Y -403.284,Z 419.585,A 0.000,B 0.000,C 90.000,E1 285.300} C_DIS
LIN {X -0.223,Y -421.525,Z 419.575,A 0.000,B 0.000,C 90.000,E1 283.536} C_DIS
LIN {X 0.103,Y -431.836,Z 419.569,A 0.000,B 0.000,C 90.000,E1 282.479} C_DIS
LIN {X 0.088,Y -439.386,Z 419.565,A 0.000,B 0.000,C 90.000,E1 281.715} C_DIS
LIN {X -0.065,Y -446.600,Z 419.561,A 0.000,B 0.000,C 90.000,E1 280.950} C_DIS
LIN {X 0.122,Y -453.348,Z 419.556,A 0.000,B 0.000,C 90.000,E1 280.141} C_DIS
LIN {X 0.200,Y -461.489,Z 419.551,A 0.000,B 0.000,C 90.000,E1 279.095} C_DIS
LIN {X 0.072,Y -467.008,Z 419.546,A 0.000,B 0.000,C 90.000,E1 278.341} C_DIS
LIN {X -0.163,Y -473.777,Z 419.541,A 0.000,B 0.000,C 90.000,E1 277.352} C_DIS
LIN {X 0.087,Y -479.857,Z 419.535,A 0.000,B 0.000,C 90.000,E1 276.315} C_DIS
LIN {X 0.062,Y -483.826,Z 419.531,A 0.000,B 0.000,C 90.000,E1 275.568} C_DIS
LIN {X 0.072,Y -487.035,Z 419.527,A 0.000,B 0.000,C 90.000,E1 274.821} C_DIS
LIN {X -0.216,Y -488.765,Z 419.524,A 0.000,B 0.000,C 90.000,E1 274.359} C_DIS
LIN {X -0.013,Y -490.122,Z 419.521,A 0.000,B 0.000,C 90.000,E1 273.841} C_DIS
LIN {X 0.167,Y -491.121,Z 419.519,A 0.000,B 0.000,C 90.000,E1 273.326} C_DIS
LIN {X -0.105,Y -491.828,Z 419.516,A 0.000,B 0.000,C 90.000,E1 272.865} C_DIS
LIN {X 0.093,Y -492.169,Z 419.513,A 0.000,B 0.000,C 90.000,E1 272.350} C_DIS
LIN {X -0.193,Y -492.114,Z 419.510,A 0.000,B 0.000,C 90.000,E1 271.892} C_DIS
LIN {X 0.028,Y -491.663,Z 419.508,A 0.000,B 0.000,C 90.000,E1 271.375} C_DIS
LIN {X 0.235,Y -490.716,Z 419.505,A 0.000,B 0.000,C 90.000,E1 270.859} C_DIS
LIN {X -0.050,Y -489.324,Z 419.502,A 0.000,B 0.000,C 90.000,E1 270.401} C_DIS
LIN {X 0.149,Y -487.364,Z 419.499,A 0.000,B 0.000,C 90.000,E1 269.885} C_DIS
LIN {X -0.146,Y -484.778,Z 419.497,A 0.000,B 0.000,C 90.000,E1 269.427} C_DIS
LIN {X 0.180,Y -483.283,Z 419.495,A 0.000,B 0.000,C 90.000,E1 269.141} C_DIS
LIN {X -0.139,Y -479.543,Z 419.493,A 0.000,B 0.000,C 90.000,E1 268.682} C_DIS
LIN {X 0.016,Y -474.873,Z 419.490,A 0.000,B 0.000,C 90.000,E1 268.165} C_DIS
LIN {X -0.158,Y -469.255,Z 419.487,A 0.000,B 0.000,C 90.000,E1 267.707} C_DIS
LIN {X -0.162,Y -466.067,Z 419.486,A 0.000,B 0.000,C 90.000,E1 267.478} C_DIS
LIN {X -0.132,Y -459.245,Z 419.484,A 0.000,B 0.000,C 90.000,E1 267.078} C_DIS
LIN {X 0.047,Y -451.895,Z 419.482,A 0.000,B 0.000,C 90.000,E1 266.731} C_DIS
LIN {X -0.164,Y -444.669,Z 419.480,A 0.000,B 0.000,C 90.000,E1 266.502} C_DIS
LIN {X 0.031,Y -437.182,Z 419.479,A 0.000,B 0.000,C 90.000,E1 266.274} C_DIS
LIN {X 0.119,Y -428.927,Z 419.478,A 0.000,B 0.000,C 90.000,E1 266.102} C_DIS
LIN {X 0.104,Y -419.384,Z 419.478,A 0.000,B 0.000,C 90.000,E1 265.988} C_DIS
LIN {X 0.158,Y -411.393,Z 419.478,A 0.000,B 0.000,C 90.000,E1 265.931} C_DIS
LIN {X 0.115,Y -406.648,Z 419.477,A 0.000,B 0.000,C 90.000,E1 265.927} C_DIS
LIN {X 0.020,Y -180.918,Z 419.477,A 0.000,B 0.000,C 90.000,E1 265.927} C_DIS
LIN {X 0.051,Y -180.839,Z 419.472,A 0.000,B 0.000,C 90.000,E1 264.894} C_DIS
LIN {X -0.052,Y -178.880,Z 419.443,A 0.000,B 0.000,C 90.000,E1 259.690} C_DIS
LIN {X 0.024,Y -175.922,Z 419.414,A 0.000,B 0.000,C 90.000,E1 254.574} C_DIS
LIN {X -0.087,Y -174.622,Z 419.405,A 0.000,B 0.000,C 90.000,E1 252.906} C_DIS
LIN {X 0.006,Y -171.602,Z 419.381,A 0.000,B 0.000,C 90.000,E1 248.592} C_DIS
LIN {X -0.005,Y -167.825,Z 419.357,A 0.000,B 0.000,C 90.000,E1 244.280} C_DIS
LIN {X 0.012,Y -166.549,Z 419.347,A 0.000,B 0.000,C 90.000,E1 242.538} C_DIS
LIN {X -0.078,Y -162.544,Z 419.323,A 0.000,B 0.000,C 90.000,E1 238.201} C_DIS
LIN {X -0.017,Y -161.222,Z 419.313,A 0.000,B 0.000,C 90.000,E1 236.421} C_DIS
LIN {X 0.018,Y -157.228,Z 419.289,A 0.000,B 0.000,C 90.000,E1 231.984} C_DIS
LIN {X 0.041,Y -155.954,Z 419.279,A 0.000,B 0.000,C 90.000,E1 230.194} C_DIS
LIN {X -0.001,Y -152.206,Z 419.254,A 0.000,B 0.000,C 90.000,E1 225.729} C_DIS
LIN {X 0.021,Y -150.452,Z 419.239,A 0.000,B 0.000,C 90.000,E1 223.014} C_DIS
LIN {X 0.048,Y -147.178,Z 419.214,A 0.000,B 0.000,C 90.000,E1 218.463} C_DIS
LIN {X 0.014,Y -145.195,Z 419.193,A 0.000,B 0.000,C 90.000,E1 214.818} C_DIS
LIN {X 0.048,Y -142.335,Z 419.163,A 0.000,B 0.000,C 90.000,E1 209.283} C_DIS
LIN {X -0.022,Y -141.724,Z 419.153,A 0.000,B 0.000,C 90.000,E1 207.462} C_DIS
LIN {X -0.040,Y -139.478,Z 419.116,A 0.000,B 0.000,C 90.000,E1 200.972} C_DIS
LIN {X -0.052,Y -138.976,Z 419.101,A 0.000,B 0.000,C 90.000,E1 198.181} C_DIS
LIN {X 0.070,Y -138.331,Z 419.054,A 0.000,B 0.000,C 90.000,E1 189.726} C_DIS
LIN {X -0.066,Y -139.432,Z 419.007,A 0.000,B 0.000,C 90.000,E1 181.375} C_DIS
LIN {X 0.014,Y -140.958,Z 418.976,A 0.000,B 0.000,C 90.000,E1 175.755} C_DIS
LIN {X -0.036,Y -142.714,Z 418.956,A 0.000,B 0.000,C 90.000,E1 172.064} C_DIS
LIN {X 0.064,Y -145.090,Z 418.930,A 0.000,B 0.000,C 90.000,E1 167.409} C_DIS
LIN {X 0.059,Y -147.715,Z 418.910,A 0.000,B 0.000,C 90.000,E1 163.740} C_DIS
LIN {X 0.000,Y -150.373,Z 418.890,A 0.000,B 0.000,C 90.000,E1 160.115} C_DIS
LIN {X 0.018,Y -153.801,Z 418.869,A 0.000,B 0.000,C 90.000,E1 156.485} C_DIS
LIN {X 0.078,Y -157.212,Z 418.849,A 0.000,B 0.000,C 90.000,E1 152.871} C_DIS
LIN {X 0.019,Y -161.377,Z 418.830,A 0.000,B 0.000,C 90.000,E1 149.331} C_DIS
LIN {X 0.030,Y -165.579,Z 418.810,A 0.000,B 0.000,C 90.000,E1 145.801} C_DIS
LIN {X 0.017,Y -170.500,Z 418.791,A 0.000,B 0.000,C 90.000,E1 142.316} C_DIS
LIN {X 0.061,Y -175.380,Z 418.772,A 0.000,B 0.000,C 90.000,E1 138.852} C_DIS
LIN {X -0.076,Y -181.003,Z 418.753,A 0.000,B 0.000,C 90.000,E1 135.486} C_DIS
LIN {X 0.049,Y -186.432,Z 418.734,A 0.000,B 0.000,C 90.000,E1 132.081} C_DIS
LIN {X 0.117,Y -191.059,Z 418.720,A 0.000,B 0.000,C 90.000,E1 129.564} C_DIS
LIN {X -0.027,Y -196.640,Z 418.702,A 0.000,B 0.000,C 90.000,E1 126.423} C_DIS
LIN {X -0.075,Y -295.530,Z 418.702,A 0.000,B 0.000,C 90.000,E1 126.423} C_DIS
LIN {X 0.061,Y -299.153,Z 418.702,A 0.000,B 0.000,C 90.000,E1 126.297} C_DIS
LIN {X 0.078,Y -302.408,Z 418.701,A 0.000,B 0.000,C 90.000,E1 126.091} C_DIS
LIN {X 0.009,Y -306.059,Z 418.698,A 0.000,B 0.000,C 90.000,E1 125.724} C_DIS
LIN {X -0.044,Y -309.575,Z 418.695,A 0.000,B 0.000,C 90.000,E1 125.152} C_DIS
LIN {X -0.012,Y -310.968,Z 418.693,A 0.000,B 0.000,C 90.000,E1 124.818} C_DIS
LIN {X 0.058,Y -323.031,Z 418.674,A 0.000,B 0.000,C 90.000,E1 121.258} C_DIS
LIN {X -0.067,Y -334.285,Z 418.658,A 0.000,B 0.000,C 90.000,E1 118.437} C_DIS
LIN {X -0.039,Y -346.970,Z 418.642,A 0.000,B 0.000,C 90.000,E1 115.643} C_DIS
LIN {X 0.018,Y -359.534,Z 418.629,A 0.000,B 0.000,C 90.000,E1 113.206} C_DIS
LIN {X -0.080,Y -373.407,Z 418.616,A 0.000,B 0.000,C 90.000,E1 110.844} C_DIS
